C07332=1142.732,180.270,-61.153,-178.357,7.250,148.882
C07333=1142.727,180.518,-61.175,-178.354,7.252,148.881
C07334=1142.723,180.767,-61.199,-178.351,7.255,148.881
C07335=1142.718,181.017,-61.221,-178.348,7.256,148.881
C07336=1142.714,181.265,-61.244,-178.346,7.259,148.881
C07337=1142.709,181.514,-61.268,-178.343,7.261,148.880
C07338=1142.704,181.763,-61.291,-178.340,7.264,148.880
C07339=1142.700,182.011,-61.313,-178.337,7.266,148.880
C07340=1142.695,182.260,-61.337,-178.334,7.268,148.879
C07341=1142.690,182.509,-61.360,-178.332,7.270,148.879
C07342=1142.686,182.758,-61.383,-178.329,7.273,148.879
C07343=1142.682,183.007,-61.406,-178.326,7.275,148.879
C07344=1142.676,183.277,-61.431,-178.323,7.277,148.878
C07345=1142.671,183.547,-61.456,-178.320,7.280,148.878
C07346=1142.666,183.817,-61.481,-178.316,7.283,148.878
C07347=1142.661,184.085,-61.506,-178.314,7.285,148.878
C07348=1142.657,184.334,-61.530,-178.311,7.287,148.877
C07349=1142.652,184.583,-61.553,-178.308,7.290,148.877
C07350=1142.647,184.832,-61.576,-178.305,7.292,148.877
C07351=1142.643,185.081,-61.600,-178.302,7.294,148.876
C07352=1142.639,185.330,-61.623,-178.300,7.296,148.876
C07353=1142.634,185.579,-61.646,-178.297,7.299,148.876
C07354=1142.629,185.828,-61.669,-178.294,7.301,148.876
C07355=1142.625,186.077,-61.693,-178.291,7.304,148.875
C07356=1142.620,186.326,-61.716,-178.289,7.306,148.875
C07357=1142.615,186.575,-61.739,-178.286,7.308,148.875
C07358=1142.612,186.823,-61.763,-178.283,7.311,148.875
C07359=1142.607,187.072,-61.786,-178.280,7.313,148.874
C07360=1142.602,187.321,-61.809,-178.277,7.315,148.874
C07361=1142.597,187.570,-61.833,-178.275,7.318,148.874
C07362=1142.592,187.819,-61.856,-178.271,7.320,148.874
C07363=1142.587,188.068,-61.879,-178.269,7.322,148.874
C07364=1142.583,188.316,-61.903,-178.266,7.325,148.873
C07365=1142.578,188.565,-61.927,-178.264,7.327,148.873
C07366=1142.574,188.814,-61.950,-178.260,7.329,148.873
C07367=1142.569,189.063,-61.973,-178.258,7.331,148.873
C07368=1142.565,189.312,-61.998,-178.255,7.334,148.872
C07369=1142.560,189.561,-62.021,-178.252,7.337,148.872
C07370=1142.555,189.810,-62.044,-178.249,7.339,148.872
C07371=1142.551,190.058,-62.068,-178.247,7.342,148.872
C07372=1142.546,190.307,-62.092,-178.244,7.343,148.871
C07373=1142.541,190.556,-62.115,-178.241,7.346,148.871
C07374=1142.537,190.805,-62.139,-178.238,7.348,148.871
C07375=1142.532,191.054,-62.162,-178.236,7.351,148.871
C07376=1142.528,191.303,-62.186,-178.232,7.353,148.870
C07377=1142.523,191.551,-62.210,-178.230,7.355,148.870
C07378=1142.518,191.800,-62.233,-178.227,7.358,148.870
C07379=1142.514,192.050,-62.257,-178.224,7.360,148.870
C07380=1142.510,192.298,-62.281,-178.221,7.363,148.869
C07381=1142.505,192.547,-62.304,-178.218,7.366,148.869
C07382=1142.501,192.796,-62.328,-178.216,7.367,148.869
C07383=1142.496,193.045,-62.352,-178.213,7.370,148.869
C07384=1142.492,193.293,-62.376,-178.210,7.372,148.868
C07385=1142.487,193.542,-62.399,-178.207,7.375,148.868
C07386=1142.482,193.791,-62.424,-178.205,7.377,148.868
C07387=1142.477,194.040,-62.447,-178.202,7.379,148.868
C07388=1142.473,194.289,-62.471,-178.199,7.382,148.868
C07389=1142.468,194.538,-62.495,-178.196,7.384,148.867
C07390=1142.464,194.786,-62.519,-178.193,7.387,148.867
C07391=1142.460,195.036,-62.543,-178.190,7.390,148.867
C07392=1142.455,195.284,-62.567,-178.188,7.391,148.867
C07393=1142.450,195.533,-62.591,-178.185,7.394,148.866
C07394=1142.445,195.782,-62.615,-178.182,7.396,148.866
C07395=1142.441,196.030,-62.639,-178.179,7.399,148.866
C07396=1142.436,196.279,-62.662,-178.176,7.401,148.866
C07397=1142.432,196.528,-62.686,-178.174,7.403,148.866
C07398=1142.428,196.777,-62.711,-178.171,7.406,148.865
C07399=1142.423,197.026,-62.735,-178.168,7.408,148.865
C07400=1142.418,197.275,-62.759,-178.166,7.411,148.865
C07401=1142.414,197.523,-62.783,-178.162,7.414,148.865
C07402=1142.409,197.772,-62.806,-178.160,7.416,148.865
C07403=1142.404,198.021,-62.831,-178.157,7.418,148.864
C07404=1142.400,198.270,-62.855,-178.154,7.421,148.864
C07405=1142.396,198.519,-62.879,-178.151,7.423,148.864
C07406=1142.391,198.767,-62.903,-178.148,7.426,148.864
C07407=1142.386,199.016,-62.927,-178.146,7.427,148.863
C07408=1142.382,199.264,-62.951,-178.143,7.430,148.863
C07409=1142.378,199.514,-62.976,-178.140,7.433,148.863
C07410=1142.372,199.763,-63.000,-178.137,7.435,148.863
C07411=1142.368,200.011,-63.024,-178.135,7.438,148.863
C07412=1142.364,200.260,-63.048,-178.131,7.440,148.862
C07413=1142.359,200.509,-63.073,-178.129,7.443,148.862
C07414=1142.355,200.758,-63.097,-178.126,7.445,148.862
C07415=1142.350,201.006,-63.121,-178.123,7.448,148.862
C07416=1142.345,201.255,-63.145,-178.121,7.450,148.862
C07417=1142.341,201.504,-63.169,-178.118,7.453,148.861
C07418=1142.337,201.753,-63.194,-178.115,7.456,148.861
C07419=1142.332,202.002,-63.218,-178.112,7.457,148.861
C07420=1142.327,202.250,-63.242,-178.109,7.460,148.861
C07421=1142.323,202.499,-63.267,-178.106,7.463,148.861
C07422=1142.318,202.748,-63.291,-178.104,7.465,148.860
C07423=1142.314,202.996,-63.315,-178.101,7.468,148.860
C07424=1142.309,203.246,-63.341,-178.098,7.470,148.860
C07425=1142.305,203.494,-63.365,-178.095,7.472,148.860
C07426=1142.300,203.743,-63.389,-178.093,7.475,148.860
C07427=1142.295,203.991,-63.413,-178.089,7.478,148.859
C07428=1142.292,204.240,-63.438,-178.087,7.480,148.859
C07429=1142.287,204.489,-63.462,-178.084,7.483,148.859
C07430=1142.282,204.737,-63.487,-178.081,7.485,148.859
C07431=1142.278,204.987,-63.512,-178.079,7.488,148.859
C07432=1142.273,205.235,-63.536,-178.076,7.490,148.858
C07433=1142.268,205.484,-63.560,-178.073,7.493,148.858
C07434=1142.264,205.733,-63.585,-178.071,7.495,148.858
C07435=1142.259,205.981,-63.610,-178.067,7.498,148.858
C07436=1142.254,206.230,-63.635,-178.064,7.501,148.858
C07437=1142.251,206.479,-63.659,-178.062,7.503,148.857
C07438=1142.245,206.728,-63.684,-178.059,7.505,148.857
C07439=1142.242,206.977,-63.708,-178.056,7.508,148.857
C07440=1142.236,207.226,-63.733,-178.053,7.511,148.857
C07441=1142.232,207.473,-63.758,-178.051,7.513,148.857
C07442=1142.228,207.723,-63.783,-178.048,7.516,148.856
C07443=1142.223,207.972,-63.807,-178.045,7.518,148.856
C07444=1142.218,208.220,-63.832,-178.042,7.520,148.856
C07445=1142.214,208.469,-63.857,-178.040,7.523,148.856
C07446=1142.210,208.717,-63.881,-178.036,7.526,148.856
C07447=1142.205,208.967,-63.906,-178.034,7.529,148.855
C07448=1142.200,209.237,-63.933,-178.031,7.532,148.855
C07449=1142.195,209.508,-63.960,-178.027,7.534,148.855
C07450=1142.190,209.778,-63.987,-178.025,7.537,148.855
C07451=1142.185,210.049,-64.015,-178.021,7.540,148.855
C07452=1142.181,210.297,-64.039,-178.019,7.543,148.855
C07453=1142.176,210.546,-64.064,-178.016,7.545,148.854
C07454=1142.171,210.795,-64.089,-178.013,7.547,148.854
C07455=1142.168,211.044,-64.114,-178.010,7.550,148.854
C07456=1142.163,211.292,-64.139,-178.008,7.552,148.854
C07457=1142.158,211.542,-64.164,-178.005,7.555,148.854
C07458=1142.154,211.789,-64.189,-178.002,7.558,148.853
C07459=1142.150,212.039,-64.214,-177.999,7.561,148.853
C07460=1142.145,212.287,-64.239,-177.996,7.562,148.853
C07461=1142.140,212.536,-64.264,-177.994,7.565,148.853
C07462=1142.136,212.784,-64.289,-177.991,7.568,148.853
C07463=1142.132,213.034,-64.314,-177.988,7.571,148.853
C07464=1142.127,213.282,-64.339,-177.985,7.573,148.852
C07465=1142.122,213.531,-64.364,-177.983,7.576,148.852
C07466=1142.117,213.779,-64.390,-177.980,7.579,148.852
C07467=1142.114,214.028,-64.414,-177.977,7.581,148.852
C07468=1142.109,214.276,-64.440,-177.974,7.583,148.852
C07469=1142.104,214.526,-64.465,-177.971,7.586,148.852
C07470=1142.099,214.774,-64.490,-177.969,7.589,148.851
C07471=1142.095,215.023,-64.515,-177.965,7.592,148.851
C07472=1142.091,215.271,-64.540,-177.963,7.595,148.851
C07473=1142.087,215.520,-64.566,-177.960,7.597,148.851
C07474=1142.082,215.769,-64.591,-177.958,7.600,148.851
C07475=1142.077,216.018,-64.616,-177.954,7.602,148.851
C07476=1142.073,216.266,-64.642,-177.952,7.605,148.850
C07477=1142.068,216.515,-64.667,-177.949,7.607,148.850
C07478=1142.064,216.764,-64.692,-177.947,7.610,148.850
C07479=1142.059,217.012,-64.718,-177.943,7.613,148.850
C07480=1142.055,217.261,-64.742,-177.940,7.615,148.850
C07481=1142.051,217.510,-64.768,-177.938,7.618,148.850
C07482=1142.046,217.758,-64.793,-177.935,7.620,148.850
C07483=1142.042,218.007,-64.819,-177.932,7.623,148.849
C07484=1142.037,218.256,-64.844,-177.929,7.626,148.849
C07485=1142.032,218.504,-64.869,-177.927,7.629,148.849
C07486=1142.028,218.753,-64.895,-177.924,7.631,148.849
C07487=1142.023,219.001,-64.921,-177.921,7.634,148.849
C07488=1142.019,219.251,-64.946,-177.918,7.636,148.849
C07489=1142.015,219.499,-64.971,-177.915,7.639,148.848
C07490=1142.010,219.748,-64.997,-177.913,7.642,148.848
C07491=1142.005,219.996,-65.022,-177.910,7.644,148.848
C07492=1142.001,220.245,-65.048,-177.907,7.647,148.848
C07493=1141.996,220.493,-65.074,-177.904,7.650,148.848
C07494=1141.992,220.742,-65.099,-177.902,7.653,148.848
C07495=1141.988,220.991,-65.125,-177.899,7.656,148.848
C07496=1141.983,221.240,-65.150,-177.896,7.658,148.847
C07497=1141.979,221.488,-65.175,-177.893,7.660,148.847
C07498=1141.974,221.737,-65.201,-177.890,7.663,148.847
C07499=1141.970,221.985,-65.227,-177.888,7.666,148.847
C07500=1141.965,222.234,-65.252,-177.885,7.669,148.847
C07501=1141.961,222.483,-65.278,-177.882,7.672,148.847
C07502=1141.956,222.732,-65.304,-177.879,7.674,148.847
C07503=1141.951,222.980,-65.330,-177.877,7.677,148.846
C07504=1141.947,223.229,-65.356,-177.874,7.680,148.846
C07505=1141.943,223.478,-65.381,-177.871,7.682,148.846
C07506=1141.939,223.727,-65.407,-177.868,7.685,148.846
C07507=1141.934,223.975,-65.433,-177.865,7.688,148.846
C07508=1141.930,224.223,-65.459,-177.863,7.690,148.846
C07509=1141.926,224.472,-65.485,-177.860,7.693,148.846
C07510=1141.921,224.721,-65.511,-177.857,7.696,148.846
C07511=1141.916,224.969,-65.536,-177.854,7.699,148.845
C07512=1141.912,225.218,-65.562,-177.851,7.701,148.845
C07513=1141.907,225.466,-65.588,-177.848,7.704,148.845
C07514=1141.903,225.715,-65.614,-177.845,7.707,148.845
C07515=1141.898,225.964,-65.640,-177.843,7.709,148.845
C07516=1141.894,226.212,-65.666,-177.840,7.712,148.845
C07517=1141.890,226.461,-65.692,-177.838,7.715,148.845
C07518=1141.885,226.710,-65.718,-177.834,7.718,148.844
C07519=1141.880,226.959,-65.744,-177.832,7.721,148.844
C07520=1141.876,227.207,-65.769,-177.829,7.723,148.844
C07521=1141.872,227.455,-65.796,-177.826,7.726,148.844
C07522=1141.867,227.704,-65.822,-177.824,7.728,148.844
C07523=1141.862,227.953,-65.848,-177.821,7.731,148.844
C07524=1141.858,228.201,-65.874,-177.818,7.734,148.844
C07525=1141.854,228.450,-65.900,-177.815,7.737,148.844
C07526=1141.849,228.698,-65.926,-177.812,7.740,148.843
C07527=1141.845,228.946,-65.953,-177.809,7.743,148.843
C07528=1141.841,229.195,-65.978,-177.807,7.746,148.843
C07529=1141.836,229.444,-66.004,-177.804,7.748,148.843
C07530=1141.832,229.693,-66.031,-177.802,7.751,148.843
C07531=1141.827,229.941,-66.057,-177.799,7.754,148.843
C07532=1141.822,230.190,-66.083,-177.796,7.756,148.843
C07533=1141.818,230.438,-66.109,-177.793,7.759,148.843
C07534=1141.814,230.687,-66.135,-177.790,7.762,148.842
C07535=1141.809,230.935,-66.162,-177.787,7.765,148.842
C07536=1141.805,231.184,-66.188,-177.784,7.768,148.842
C07537=1141.801,231.432,-66.214,-177.781,7.771,148.842
C07538=1141.796,231.681,-66.241,-177.779,7.773,148.842
C07539=1141.792,231.930,-66.266,-177.776,7.776,148.842
C07540=1141.787,232.179,-66.294,-177.774,7.779,148.842
C07541=1141.783,232.427,-66.320,-177.771,7.782,148.842
C07542=1141.778,232.676,-66.346,-177.768,7.784,148.842
C07543=1141.774,232.924,-66.373,-177.765,7.787,148.841
C07544=1141.769,233.173,-66.399,-177.762,7.790,148.841
C07545=1141.765,233.421,-66.425,-177.759,7.793,148.841
C07546=1141.761,233.670,-66.451,-177.756,7.796,148.841
C07547=1141.756,233.918,-66.478,-177.754,7.799,148.841
C07548=1141.752,234.167,-66.504,-177.751,7.801,148.841
C07549=1141.747,234.415,-66.531,-177.749,7.804,148.841
C07550=1141.743,234.663,-66.557,-177.746,7.807,148.841
C07551=1141.738,234.913,-66.584,-177.743,7.810,148.841
C07552=1141.734,235.185,-66.613,-177.740,7.812,148.841
C07553=1141.729,235.456,-66.642,-177.736,7.816,148.840
C07554=1141.724,235.728,-66.671,-177.734,7.819,148.840
C07555=1141.719,236.000,-66.700,-177.731,7.822,148.840
C07556=1141.715,236.248,-66.727,-177.728,7.825,148.840
C07557=1141.710,236.497,-66.754,-177.725,7.827,148.840
C07558=1141.705,236.746,-66.780,-177.722,7.830,148.840
C07559=1141.701,236.994,-66.807,-177.720,7.833,148.840
C07560=1141.697,237.242,-66.834,-177.717,7.836,148.840
C07561=1141.693,237.491,-66.860,-177.714,7.839,148.840
C07562=1141.689,237.740,-66.887,-177.711,7.842,148.840
C07563=1141.684,237.989,-66.914,-177.708,7.845,148.840
C07564=1141.680,238.237,-66.940,-177.706,7.848,148.840
C07565=1141.675,238.486,-66.967,-177.702,7.850,148.839
C07566=1141.670,238.734,-66.994,-177.700,7.853,148.839
C07567=1141.667,238.982,-67.021,-177.697,7.856,148.839
C07568=1141.662,239.231,-67.048,-177.695,7.858,148.839
C07569=1141.657,239.480,-67.074,-177.692,7.861,148.839
C07570=1141.653,239.728,-67.101,-177.689,7.864,148.839
C07571=1141.648,239.977,-67.128,-177.686,7.867,148.839
C07572=1141.644,240.225,-67.155,-177.683,7.870,148.839
C07573=1141.639,240.474,-67.182,-177.681,7.873,148.839
C07574=1141.635,240.722,-67.208,-177.678,7.876,148.838
C07575=1141.631,240.971,-67.236,-177.675,7.879,148.838
C07576=1141.626,241.220,-67.263,-177.672,7.882,148.838
C07577=1141.622,241.468,-67.289,-177.669,7.885,148.838
C07578=1141.618,241.716,-67.316,-177.667,7.888,148.838
C07579=1141.613,241.965,-67.343,-177.664,7.890,148.838
C07580=1141.608,242.213,-67.371,-177.661,7.893,148.838
C07581=1141.604,242.462,-67.398,-177.658,7.896,148.838
C07582=1141.601,242.711,-67.424,-177.655,7.899,148.838
C07583=1141.596,242.959,-67.451,-177.653,7.902,148.838
C07584=1141.591,243.207,-67.479,-177.650,7.905,148.838
C07585=1141.587,243.455,-67.506,-177.647,7.908,148.838
C07586=1141.582,243.704,-67.533,-177.644,7.911,148.838
C07587=1141.578,243.952,-67.560,-177.641,7.914,148.837
C07588=1141.574,244.201,-67.587,-177.639,7.917,148.837
C07589=1141.570,244.450,-67.614,-177.636,7.920,148.837
C07590=1141.565,244.698,-67.641,-177.633,7.923,148.837
C07591=1141.561,244.946,-67.669,-177.630,7.925,148.837
C07592=1141.556,245.195,-67.696,-177.627,7.928,148.837
C07593=1141.552,245.444,-67.724,-177.625,7.931,148.837
C07594=1141.547,245.692,-67.751,-177.622,7.934,148.837
C07595=1141.543,245.940,-67.779,-177.619,7.937,148.837
C07596=1141.538,246.189,-67.806,-177.616,7.940,148.837
C07597=1141.534,246.437,-67.832,-177.613,7.943,148.837
C07598=1141.530,246.686,-67.859,-177.611,7.946,148.837
C07599=1141.526,246.934,-67.887,-177.608,7.949,148.837
C07600=1141.521,247.182,-67.914,-177.606,7.952,148.837
C07601=1141.517,247.431,-67.941,-177.603,7.955,148.837
C07602=1141.513,247.680,-67.970,-177.600,7.958,148.837
C07603=1141.508,247.928,-67.997,-177.597,7.961,148.836
C07604=1141.503,248.177,-68.024,-177.594,7.964,148.836
C07605=1141.499,248.424,-68.051,-177.592,7.967,148.836
C07606=1141.495,248.674,-68.079,-177.589,7.970,148.836
C07607=1141.491,248.921,-68.107,-177.586,7.973,148.836
C07608=1141.486,249.170,-68.134,-177.583,7.975,148.836
C07609=1141.482,249.419,-68.161,-177.580,7.978,148.836
C07610=1141.478,249.667,-68.189,-177.578,7.981,148.836
C07611=1141.473,249.916,-68.216,-177.575,7.984,148.836
C07612=1141.469,250.164,-68.245,-177.572,7.987,148.836
C07613=1141.464,250.413,-68.272,-177.569,7.990,148.836
C07614=1141.459,250.661,-68.300,-177.566,7.993,148.836
C07615=1141.455,250.910,-68.327,-177.564,7.996,148.836
C07616=1141.451,251.158,-68.355,-177.561,7.999,148.836
C07617=1141.446,251.406,-68.382,-177.558,8.002,148.836
C07618=1141.443,251.655,-68.410,-177.556,8.005,148.836
C07619=1141.438,251.903,-68.438,-177.553,8.008,148.836
C07620=1141.434,252.151,-68.465,-177.550,8.011,148.835
C07621=1141.430,252.400,-68.493,-177.547,8.014,148.835
C07622=1141.425,252.649,-68.521,-177.545,8.017,148.835
C07623=1141.420,252.897,-68.548,-177.542,8.020,148.835
C07624=1141.416,253.145,-68.576,-177.539,8.022,148.835
C07625=1141.412,253.394,-68.604,-177.536,8.025,148.835
C07626=1141.408,253.642,-68.632,-177.533,8.028,148.835
C07627=1141.403,253.890,-68.660,-177.531,8.032,148.835
C07628=1141.398,254.139,-68.687,-177.528,8.035,148.835
C07629=1141.395,254.388,-68.715,-177.525,8.037,148.835
C07630=1141.390,254.635,-68.743,-177.523,8.040,148.835
C07631=1141.386,254.884,-68.771,-177.520,8.043,148.835
C07632=1141.381,255.133,-68.799,-177.517,8.046,148.835
C07633=1141.377,255.381,-68.827,-177.514,8.050,148.835
C07634=1141.373,255.629,-68.855,-177.511,8.053,148.835
C07635=1141.369,255.877,-68.883,-177.509,8.056,148.835
C07636=1141.364,256.127,-68.911,-177.506,8.059,148.835
C07637=1141.359,256.374,-68.938,-177.503,8.062,148.835
C07638=1141.356,256.623,-68.966,-177.500,8.065,148.835
C07639=1141.351,256.871,-68.995,-177.497,8.068,148.835
C07640=1141.347,257.120,-69.023,-177.495,8.071,148.835
C07641=1141.343,257.368,-69.051,-177.492,8.074,148.834
C07642=1141.338,257.617,-69.080,-177.489,8.077,148.835
C07643=1141.334,257.864,-69.107,-177.487,8.080,148.835
C07644=1141.330,258.114,-69.135,-177.484,8.083,148.834
C07645=1141.325,258.362,-69.163,-177.481,8.086,148.834
C07646=1141.321,258.610,-69.191,-177.478,8.089,148.834
C07647=1141.316,258.858,-69.219,-177.475,8.092,148.834
C07648=1141.312,259.107,-69.248,-177.472,8.095,148.834
C07649=1141.308,259.355,-69.276,-177.470,8.099,148.834
C07650=1141.303,259.604,-69.304,-177.467,8.101,148.834
C07651=1141.299,259.852,-69.332,-177.464,8.104,148.834
C07652=1141.295,260.100,-69.360,-177.461,8.107,148.834
C07653=1141.290,260.349,-69.389,-177.459,8.110,148.834
C07654=1141.286,260.597,-69.417,-177.456,8.113,148.834
C07655=1141.281,260.845,-69.445,-177.453,8.116,148.834
C07656=1141.277,261.119,-69.477,-177.450,8.120,148.834
C07657=1141.272,261.392,-69.508,-177.447,8.123,148.834
C07658=1141.267,261.666,-69.539,-177.444,8.127,148.834
C07659=1141.262,261.939,-69.570,-177.441,8.130,148.834
C07660=1141.258,262.187,-69.599,-177.438,8.133,148.834
C07661=1141.254,262.436,-69.628,-177.436,8.136,148.834
C07662=1141.250,262.684,-69.655,-177.433,8.139,148.834
C07663=1141.245,262.933,-69.684,-177.430,8.143,148.834
C07664=1141.241,263.181,-69.712,-177.427,8.145,148.834
C07665=1141.237,263.429,-69.741,-177.424,8.148,148.834
C07666=1141.233,263.678,-69.770,-177.422,8.152,148.834
C07667=1141.228,263.926,-69.798,-177.419,8.155,148.834
C07668=1141.224,264.174,-69.826,-177.416,8.157,148.834
C07669=1141.219,264.423,-69.854,-177.414,8.160,148.834
C07670=1141.215,264.671,-69.884,-177.411,8.163,148.834
C07671=1141.211,264.920,-69.912,-177.408,8.167,148.834
C07672=1141.206,265.168,-69.940,-177.405,8.170,148.834
C07673=1141.202,265.416,-69.969,-177.402,8.173,148.834
C07674=1141.198,265.665,-69.998,-177.399,8.176,148.834
C07675=1141.193,265.913,-70.026,-177.397,8.179,148.834
C07676=1141.189,266.161,-70.055,-177.394,8.182,148.834
C07677=1141.185,266.410,-70.084,-177.392,8.185,148.834
C07678=1141.180,266.657,-70.113,-177.389,8.188,148.834
C07679=1141.176,266.906,-70.141,-177.386,8.191,148.834
C07680=1141.172,267.155,-70.170,-177.383,8.195,148.834
C07681=1141.167,267.402,-70.199,-177.380,8.198,148.834
C07682=1141.163,267.651,-70.227,-177.377,8.201,148.834
C07683=1141.159,267.899,-70.257,-177.375,8.204,148.834
C07684=1141.155,268.148,-70.285,-177.372,8.207,148.834
C07685=1141.150,268.395,-70.314,-177.370,8.210,148.834
C07686=1141.146,268.644,-70.343,-177.367,8.213,148.834
C07687=1141.142,268.892,-70.372,-177.364,8.217,148.834
C07688=1141.137,269.140,-70.400,-177.361,8.220,148.834
C07689=1141.133,269.388,-70.429,-177.358,8.223,148.834
C07690=1141.129,269.637,-70.458,-177.356,8.226,148.834
C07691=1141.125,269.886,-70.487,-177.353,8.229,148.834
C07692=1141.120,270.133,-70.517,-177.350,8.232,148.834
C07693=1141.115,270.382,-70.545,-177.348,8.235,148.834
C07694=1141.112,270.630,-70.574,-177.345,8.239,148.834
C07695=1141.108,270.879,-70.603,-177.342,8.242,148.834
C07696=1141.103,271.126,-70.632,-177.339,8.245,148.834
C07697=1141.099,271.375,-70.661,-177.337,8.248,148.834
C07698=1141.094,271.624,-70.690,-177.334,8.251,148.834
C07699=1141.090,271.872,-70.720,-177.331,8.254,148.834
C07700=1141.086,272.120,-70.748,-177.328,8.258,148.834
C07701=1141.081,272.368,-70.777,-177.325,8.261,148.834
C07702=1141.077,272.616,-70.806,-177.323,8.264,148.834
C07703=1141.073,272.865,-70.836,-177.320,8.267,148.834
C07704=1141.069,273.113,-70.865,-177.318,8.270,148.834
C07705=1141.064,273.362,-70.894,-177.315,8.273,148.834
C07706=1141.060,273.610,-70.923,-177.311,8.277,148.834
C07707=1141.055,273.858,-70.952,-177.309,8.280,148.834
C07708=1141.051,274.106,-70.982,-177.306,8.283,148.834
C07709=1141.048,274.354,-71.011,-177.303,8.286,148.834
C07710=1141.044,274.602,-71.040,-177.301,8.289,148.834
C07711=1141.039,274.851,-71.069,-177.298,8.292,148.834
C07712=1141.035,275.099,-71.098,-177.295,8.296,148.834
C07713=1141.031,275.347,-71.128,-177.293,8.299,148.834
C07714=1141.027,275.596,-71.157,-177.290,8.302,148.834
C07715=1141.022,275.843,-71.186,-177.288,8.305,148.834
C07716=1141.018,276.092,-71.216,-177.285,8.308,148.834
C07717=1141.013,276.340,-71.245,-177.281,8.312,148.834
C07718=1141.009,276.588,-71.275,-177.279,8.315,148.835
C07719=1141.005,276.836,-71.304,-177.276,8.318,148.835
C07720=1141.001,277.085,-71.334,-177.273,8.321,148.834
C07721=1140.997,277.333,-71.363,-177.271,8.324,148.835
C07722=1140.992,277.581,-71.393,-177.268,8.328,148.835
C07723=1140.988,277.829,-71.422,-177.265,8.331,148.835
C07724=1140.984,278.078,-71.452,-177.263,8.334,148.835
C07725=1140.979,278.326,-71.482,-177.260,8.337,148.835
C07726=1140.975,278.575,-71.511,-177.257,8.340,148.835
C07727=1140.971,278.823,-71.540,-177.254,8.344,148.835
C07728=1140.966,279.070,-71.570,-177.251,8.347,148.835
C07729=1140.962,279.319,-71.599,-177.249,8.350,148.835
C07730=1140.958,279.567,-71.628,-177.246,8.353,148.835
C07731=1140.954,279.815,-71.659,-177.244,8.357,148.835
C07732=1140.950,280.063,-71.688,-177.240,8.360,148.835
C07733=1140.945,280.311,-71.718,-177.238,8.363,148.835
C07734=1140.941,280.560,-71.748,-177.235,8.367,148.835
C07735=1140.936,280.808,-71.777,-177.233,8.369,148.835
C07736=1140.932,281.056,-71.806,-177.230,8.373,148.835
C07737=1140.928,281.304,-71.837,-177.227,8.376,148.835
C07738=1140.924,281.552,-71.866,-177.225,8.380,148.835
C07739=1140.919,281.801,-71.896,-177.222,8.383,148.835
C07740=1140.915,282.049,-71.926,-177.219,8.386,148.835
C07741=1140.911,282.297,-71.956,-177.216,8.390,148.835
C07742=1140.907,282.545,-71.985,-177.213,8.393,148.835
C07743=1140.902,282.793,-72.015,-177.211,8.396,148.836
C07744=1140.898,283.041,-72.045,-177.208,8.399,148.836
C07745=1140.895,283.290,-72.075,-177.205,8.403,148.836
C07746=1140.890,283.538,-72.105,-177.202,8.406,148.836
C07747=1140.886,283.786,-72.135,-177.200,8.409,148.836
C07748=1140.882,284.035,-72.165,-177.197,8.412,148.836
C07749=1140.877,284.283,-72.194,-177.195,8.415,148.836
C07750=1140.873,284.531,-72.225,-177.192,8.419,148.836
C07751=1140.869,284.779,-72.255,-177.189,8.422,148.836
C07752=1140.865,285.027,-72.285,-177.186,8.425,148.836
C07753=1140.860,285.275,-72.315,-177.184,8.428,148.836
C07754=1140.856,285.523,-72.345,-177.181,8.432,148.836
C07755=1140.852,285.771,-72.374,-177.178,8.435,148.836
C07756=1140.847,286.019,-72.405,-177.176,8.438,148.836
C07757=1140.844,286.268,-72.435,-177.173,8.441,148.836
C07758=1140.840,286.516,-72.465,-177.170,8.445,148.837
C07759=1140.835,286.764,-72.495,-177.167,8.448,148.836
C07760=1140.830,287.039,-72.529,-177.164,8.452,148.837
C07761=1140.825,287.316,-72.562,-177.161,8.455,148.837
C07762=1140.820,287.590,-72.595,-177.159,8.459,148.837
C07763=1140.816,287.866,-72.629,-177.155,8.463,148.837
C07764=1140.811,288.114,-72.659,-177.153,8.466,148.837
C07765=1140.808,288.362,-72.689,-177.150,8.469,148.837
C07766=1140.804,288.611,-72.720,-177.147,8.473,148.837
C07767=1140.799,288.859,-72.750,-177.144,8.476,148.837
C07768=1140.795,289.107,-72.781,-177.142,8.480,148.837
C07769=1140.791,289.355,-72.811,-177.139,8.483,148.837
C07770=1140.786,289.603,-72.841,-177.136,8.487,148.837
C07771=1140.783,289.851,-72.871,-177.133,8.489,148.837
C07772=1140.778,290.099,-72.902,-177.131,8.493,148.838
C07773=1140.774,290.348,-72.932,-177.128,8.496,148.838
C07774=1140.769,290.596,-72.962,-177.125,8.500,148.838
C07775=1140.765,290.843,-72.993,-177.123,8.503,148.838
C07776=1140.761,291.092,-73.024,-177.120,8.507,148.838
C07777=1140.758,291.340,-73.054,-177.117,8.510,148.838
C07778=1140.753,291.588,-73.084,-177.115,8.513,148.838
C07779=1140.749,291.836,-73.114,-177.112,8.516,148.838
C07780=1140.745,292.084,-73.145,-177.109,8.520,148.838
C07781=1140.741,292.332,-73.175,-177.107,8.523,148.838
C07782=1140.736,292.580,-73.206,-177.104,8.526,148.839
C07783=1140.732,292.828,-73.237,-177.101,8.530,148.839
C07784=1140.728,293.076,-73.267,-177.099,8.533,148.839
C07785=1140.723,293.325,-73.298,-177.096,8.536,148.839
C07786=1140.719,293.573,-73.328,-177.093,8.540,148.839
C07787=1140.715,293.821,-73.358,-177.090,8.544,148.839
C07788=1140.711,294.069,-73.390,-177.088,8.547,148.839
C07789=1140.707,294.317,-73.420,-177.085,8.550,148.839
C07790=1140.702,294.565,-73.451,-177.082,8.554,148.839
C07791=1140.698,294.814,-73.482,-177.080,8.557,148.839
C07792=1140.695,295.061,-73.512,-177.077,8.560,148.840
C07793=1140.690,295.309,-73.543,-177.074,8.564,148.840
C07794=1140.686,295.558,-73.574,-177.072,8.567,148.840
C07795=1140.681,295.806,-73.604,-177.069,8.570,148.840
C07796=1140.677,296.053,-73.635,-177.066,8.574,148.840
C07797=1140.674,296.301,-73.666,-177.064,8.577,148.840
C07798=1140.669,296.549,-73.697,-177.061,8.580,148.840
C07799=1140.665,296.797,-73.727,-177.058,8.584,148.840
C07800=1140.661,297.046,-73.759,-177.056,8.588,148.840
C07801=1140.657,297.294,-73.789,-177.053,8.591,148.840
C07802=1140.653,297.542,-73.820,-177.050,8.595,148.841
C07803=1140.648,297.790,-73.851,-177.047,8.598,148.841
C07804=1140.644,298.037,-73.882,-177.045,8.601,148.841
C07805=1140.640,298.286,-73.913,-177.042,8.605,148.841
C07806=1140.636,298.534,-73.944,-177.039,8.608,148.841
C07807=1140.631,298.782,-73.975,-177.037,8.611,148.841
C07808=1140.627,299.031,-74.006,-177.034,8.615,148.841
C07809=1140.623,299.278,-74.037,-177.031,8.619,148.841
C07810=1140.620,299.526,-74.068,-177.029,8.621,148.841
C07811=1140.615,299.774,-74.099,-177.026,8.626,148.842
C07812=1140.611,300.021,-74.130,-177.023,8.629,148.842
C07813=1140.607,300.270,-74.161,-177.021,8.632,148.842
C07814=1140.602,300.518,-74.192,-177.018,8.636,148.842
C07815=1140.598,300.766,-74.224,-177.015,8.639,148.842
C07816=1140.594,301.014,-74.255,-177.013,8.642,148.842
C07817=1140.590,301.263,-74.286,-177.010,8.646,148.842
C07818=1140.585,301.510,-74.317,-177.007,8.649,148.842
C07819=1140.581,301.759,-74.348,-177.004,8.653,148.843
C07820=1140.577,302.007,-74.379,-177.002,8.656,148.843
C07821=1140.574,302.254,-74.410,-176.999,8.660,148.843
C07822=1140.569,302.502,-74.441,-176.996,8.664,148.843
C07823=1140.565,302.750,-74.473,-176.994,8.667,148.843
C07824=1140.561,302.998,-74.504,-176.991,8.670,148.843
C07825=1140.557,303.246,-74.535,-176.988,8.674,148.843
C07826=1140.553,303.494,-74.566,-176.986,8.677,148.844
C07827=1140.548,303.742,-74.598,-176.983,8.681,148.844
C07828=1140.544,303.991,-74.630,-176.980,8.684,148.844
C07829=1140.539,304.238,-74.661,-176.978,8.687,148.844
C07830=1140.535,304.487,-74.692,-176.975,8.692,148.844
C07831=1140.531,304.734,-74.724,-176.973,8.695,148.844
C07832=1140.527,304.983,-74.755,-176.970,8.698,148.844
C07833=1140.523,305.231,-74.787,-176.967,8.702,148.845
C07834=1140.519,305.478,-74.818,-176.965,8.705,148.845
C07835=1140.515,305.727,-74.849,-176.962,8.709,148.845
C07836=1140.511,305.974,-74.881,-176.959,8.712,148.845
C07837=1140.507,306.222,-74.913,-176.956,8.715,148.845
C07838=1140.502,306.470,-74.943,-176.954,8.719,148.845
C07839=1140.499,306.718,-74.975,-176.951,8.723,148.845
C07840=1140.493,306.966,-75.007,-176.948,8.727,148.846
C07841=1140.489,307.214,-75.038,-176.946,8.730,148.846
C07842=1140.486,307.462,-75.070,-176.943,8.733,148.846
C07843=1140.481,307.710,-75.102,-176.940,8.737,148.846
C07844=1140.478,307.958,-75.134,-176.938,8.740,148.846
C07845=1140.473,308.206,-75.164,-176.935,8.744,148.846
C07846=1140.469,308.454,-75.197,-176.932,8.747,148.846
C07847=1140.465,308.702,-75.229,-176.930,8.751,148.847
C07848=1140.461,308.950,-75.260,-176.927,8.755,148.847
C07849=1140.457,309.198,-75.292,-176.925,8.758,148.847
C07850=1140.452,309.446,-75.323,-176.922,8.762,148.847
C07851=1140.448,309.694,-75.355,-176.919,8.765,148.847
C07852=1140.444,309.942,-75.387,-176.917,8.768,148.847
C07853=1140.440,310.189,-75.418,-176.914,8.772,148.848
C07854=1140.436,310.437,-75.450,-176.911,8.775,148.848
C07855=1140.432,310.686,-75.483,-176.908,8.780,148.848
C07856=1140.427,310.933,-75.514,-176.906,8.783,148.848
C07857=1140.424,311.181,-75.546,-176.903,8.787,148.848
C07858=1140.419,311.429,-75.579,-176.901,8.790,148.849
C07859=1140.415,311.677,-75.610,-176.898,8.793,148.849
C07860=1140.411,311.925,-75.642,-176.895,8.797,148.849
C07861=1140.408,312.173,-75.674,-176.893,8.800,148.849
C07862=1140.403,312.421,-75.706,-176.890,8.804,148.849
C07863=1140.399,312.668,-75.738,-176.887,8.808,148.849
C07864=1140.394,312.946,-75.774,-176.885,8.812,148.850
C07865=1140.390,313.225,-75.810,-176.882,8.816,148.850
C07866=1140.385,313.503,-75.845,-176.879,8.820,148.850
C07867=1140.380,313.781,-75.881,-176.876,8.824,148.850
C07868=1140.377,314.029,-75.913,-176.873,8.828,148.850
C07869=1140.372,314.276,-75.946,-176.870,8.831,148.850
C07870=1140.368,314.524,-75.977,-176.868,8.834,148.851
C07871=1140.364,314.772,-76.010,-176.865,8.838,148.851
C07872=1140.360,315.020,-76.042,-176.862,8.842,148.851
C07873=1140.356,315.268,-76.074,-176.860,8.846,148.851
C07874=1140.352,315.515,-76.106,-176.857,8.849,148.851
C07875=1140.348,315.763,-76.138,-176.854,8.853,148.852
C07876=1140.343,316.011,-76.171,-176.852,8.856,148.852
C07877=1140.340,316.260,-76.202,-176.849,8.860,148.852
C07878=1140.335,316.507,-76.234,-176.847,8.864,148.852
C07879=1140.331,316.755,-76.267,-176.844,8.868,148.852
C07880=1140.327,317.003,-76.299,-176.841,8.871,148.853
C07881=1140.323,317.251,-76.331,-176.839,8.874,148.853
C07882=1140.319,317.499,-76.364,-176.836,8.878,148.853
C07883=1140.315,317.747,-76.396,-176.834,8.882,148.853
C07884=1140.310,317.994,-76.428,-176.831,8.886,148.853
C07885=1140.307,318.242,-76.461,-176.829,8.889,148.854
C07886=1140.302,318.490,-76.493,-176.826,8.893,148.854
C07887=1140.299,318.738,-76.526,-176.823,8.896,148.854
C07888=1140.295,318.986,-76.558,-176.820,8.900,148.854
C07889=1140.290,319.234,-76.591,-176.818,8.904,148.854
C07890=1140.286,319.481,-76.623,-176.815,8.908,148.855
C07891=1140.282,319.729,-76.655,-176.813,8.911,148.855
C07892=1140.278,319.977,-76.688,-176.810,8.915,148.855
C07893=1140.274,320.225,-76.720,-176.807,8.918,148.855
C07894=1140.270,320.473,-76.754,-176.805,8.922,148.856
C07895=1140.266,320.721,-76.785,-176.802,8.926,148.856
C07896=1140.262,320.969,-76.819,-176.799,8.930,148.856
C07897=1140.258,321.217,-76.850,-176.797,8.933,148.856
C07898=1140.254,321.464,-76.884,-176.794,8.937,148.856
C07899=1140.250,321.713,-76.916,-176.792,8.940,148.857
C07900=1140.246,321.960,-76.949,-176.789,8.944,148.857
C07901=1140.241,322.207,-76.981,-176.786,8.948,148.857
C07902=1140.237,322.456,-77.014,-176.783,8.952,148.857
C07903=1140.234,322.703,-77.046,-176.781,8.955,148.857
C07904=1140.229,322.951,-77.080,-176.778,8.959,148.858
C07905=1140.225,323.199,-77.112,-176.776,8.962,148.858
C07906=1140.221,323.447,-77.145,-176.773,8.966,148.858
C07907=1140.217,323.694,-77.178,-176.771,8.970,148.858
C07908=1140.213,323.943,-77.210,-176.768,8.974,148.859
C07909=1140.209,324.190,-77.243,-176.766,8.977,148.859
C07910=1140.205,324.438,-77.277,-176.763,8.981,148.859
C07911=1140.201,324.686,-77.308,-176.760,8.984,148.859
C07912=1140.197,324.934,-77.342,-176.758,8.989,148.860
C07913=1140.193,325.181,-77.375,-176.755,8.992,148.860
C07914=1140.189,325.429,-77.408,-176.752,8.996,148.860
C07915=1140.185,325.677,-77.441,-176.750,8.999,148.860
C07916=1140.181,325.925,-77.473,-176.747,9.003,148.860
C07917=1140.177,326.173,-77.506,-176.745,9.006,148.861
C07918=1140.173,326.420,-77.539,-176.742,9.011,148.861
C07919=1140.168,326.668,-77.572,-176.739,9.015,148.861
C07920=1140.164,326.916,-77.605,-176.737,9.018,148.861
C07921=1140.160,327.164,-77.639,-176.734,9.022,148.862
C07922=1140.156,327.411,-77.672,-176.732,9.026,148.862
C07923=1140.153,327.659,-77.704,-176.729,9.030,148.862
C07924=1140.148,327.907,-77.737,-176.726,9.033,148.862
C07925=1140.144,328.154,-77.771,-176.724,9.037,148.863
C07926=1140.140,328.403,-77.803,-176.722,9.041,148.863
C07927=1140.136,328.651,-77.837,-176.719,9.045,148.863
C07928=1140.132,328.899,-77.870,-176.716,9.048,148.863
C07929=1140.128,329.146,-77.903,-176.713,9.052,148.864
C07930=1140.124,329.394,-77.936,-176.710,9.056,148.864
C07931=1140.120,329.641,-77.970,-176.708,9.060,148.864
C07932=1140.116,329.889,-78.003,-176.706,9.064,148.864
C07933=1140.112,330.137,-78.036,-176.703,9.067,148.865
C07934=1140.108,330.385,-78.069,-176.700,9.071,148.865
C07935=1140.104,330.632,-78.103,-176.698,9.074,148.865
C07936=1140.099,330.880,-78.136,-176.695,9.079,148.865
C07937=1140.095,331.128,-78.169,-176.693,9.083,148.866
C07938=1140.092,331.376,-78.202,-176.690,9.086,148.866
C07939=1140.088,331.624,-78.236,-176.687,9.090,148.866
C07940=1140.084,331.871,-78.269,-176.685,9.093,148.866
C07941=1140.080,332.119,-78.303,-176.682,9.098,148.867
C07942=1140.075,332.366,-78.336,-176.680,9.101,148.867
C07943=1140.071,332.614,-78.369,-176.677,9.105,148.867
C07944=1140.068,332.863,-78.402,-176.674,9.109,148.867
C07945=1140.064,333.110,-78.436,-176.672,9.113,148.868
C07946=1140.060,333.357,-78.469,-176.669,9.117,148.868
C07947=1140.055,333.605,-78.503,-176.667,9.120,148.868
C07948=1140.051,333.853,-78.537,-176.664,9.124,148.868
C07949=1140.047,334.100,-78.570,-176.662,9.128,148.869
C07950=1140.043,334.349,-78.604,-176.659,9.132,148.869
C07951=1140.040,334.596,-78.638,-176.656,9.136,148.869
C07952=1140.035,334.844,-78.671,-176.654,9.139,148.870
C07953=1140.031,335.091,-78.704,-176.652,9.143,148.870
C07954=1140.027,335.339,-78.738,-176.649,9.147,148.870
C07955=1140.023,335.587,-78.772,-176.646,9.151,148.870
C07956=1140.019,335.835,-78.805,-176.644,9.155,148.871
C07957=1140.015,336.082,-78.839,-176.641,9.158,148.871
C07958=1140.011,336.330,-78.872,-176.638,9.162,148.871
C07959=1140.007,336.578,-78.907,-176.636,9.166,148.872
C07960=1140.003,336.826,-78.940,-176.634,9.170,148.872
C07961=1139.999,337.073,-78.974,-176.631,9.174,148.872
C07962=1139.995,337.320,-79.007,-176.628,9.177,148.872
C07963=1139.991,337.569,-79.042,-176.626,9.182,148.873
C07964=1139.987,337.816,-79.075,-176.624,9.185,148.873
C07965=1139.983,338.063,-79.109,-176.621,9.189,148.873
C07966=1139.980,338.312,-79.142,-176.618,9.194,148.874
C07967=1139.975,338.559,-79.177,-176.616,9.197,148.874
C07968=1139.971,338.840,-79.215,-176.612,9.202,148.874
C07969=1139.966,339.120,-79.253,-176.610,9.206,148.875
C07970=1139.962,339.401,-79.292,-176.607,9.210,148.875
C07971=1139.957,339.681,-79.330,-176.604,9.215,148.875
C07972=1139.954,339.929,-79.365,-176.601,9.219,148.876
C07973=1139.949,340.177,-79.398,-176.598,9.223,148.876
C07974=1139.945,340.424,-79.432,-176.597,9.226,148.876
C07975=1139.941,340.672,-79.467,-176.594,9.230,148.876
C07976=1139.937,340.920,-79.500,-176.592,9.234,148.877
C07977=1139.933,341.167,-79.534,-176.589,9.238,148.877
C07978=1139.929,341.415,-79.569,-176.586,9.242,148.877
C07979=1139.925,341.662,-79.603,-176.584,9.246,148.878
C07980=1139.920,341.911,-79.636,-176.581,9.250,148.878
C07981=1139.917,342.158,-79.671,-176.578,9.254,148.878
C07982=1139.912,342.406,-79.705,-176.576,9.257,148.879
C07983=1139.909,342.653,-79.739,-176.573,9.261,148.879
C07984=1139.905,342.901,-79.773,-176.571,9.266,148.879
C07985=1139.900,343.149,-79.807,-176.568,9.269,148.880
C07986=1139.897,343.397,-79.841,-176.566,9.273,148.880
C07987=1139.893,343.644,-79.876,-176.563,9.278,148.880
C07988=1139.889,343.891,-79.910,-176.561,9.281,148.880
C07989=1139.885,344.139,-79.944,-176.558,9.285,148.881
C07990=1139.881,344.386,-79.978,-176.555,9.289,148.881
C07991=1139.877,344.634,-80.013,-176.553,9.293,148.882
C07992=1139.872,344.882,-80.048,-176.550,9.297,148.882
C07993=1139.869,345.130,-80.082,-176.548,9.301,148.882
C07994=1139.865,345.377,-80.116,-176.545,9.305,148.882
C07995=1139.861,345.624,-80.150,-176.543,9.309,148.883
C07996=1139.857,345.872,-80.185,-176.540,9.313,148.883
C07997=1139.853,346.119,-80.219,-176.538,9.317,148.884
C07998=1139.849,346.368,-80.254,-176.535,9.321,148.884
C07999=1139.845,346.615,-80.288,-176.532,9.325,148.884
C08000=1139.841,346.863,-80.322,-176.530,9.328,148.884
C08001=1139.837,347.110,-80.357,-176.527,9.332,148.885
C08002=1139.833,347.358,-80.391,-176.525,9.337,148.885
C08003=1139.829,347.605,-80.426,-176.523,9.340,148.885
C08004=1139.825,347.854,-80.460,-176.520,9.344,148.886
C08005=1139.821,348.100,-80.495,-176.517,9.349,148.886
C08006=1139.817,348.348,-80.530,-176.515,9.352,148.886
C08007=1139.813,348.596,-80.564,-176.512,9.356,148.887
C08008=1139.810,348.843,-80.599,-176.510,9.361,148.887
C08009=1139.805,349.091,-80.633,-176.508,9.364,148.888
C08010=1139.801,349.338,-80.669,-176.505,9.368,148.888
C08011=1139.798,349.585,-80.702,-176.502,9.373,148.888
C08012=1139.794,349.834,-80.737,-176.499,9.377,148.888
C08013=1139.789,350.081,-80.772,-176.498,9.380,148.889
C08014=1139.785,350.328,-80.807,-176.495,9.384,148.889
C08015=1139.782,350.576,-80.842,-176.492,9.389,148.890
C08016=1139.778,350.824,-80.876,-176.490,9.392,148.890
C08017=1139.774,351.071,-80.912,-176.487,9.396,148.890
C08018=1139.769,351.319,-80.946,-176.484,9.400,148.890
C08019=1139.766,351.566,-80.980,-176.482,9.405,148.891
C08020=1139.762,351.813,-81.015,-176.480,9.408,148.891
C08021=1139.758,352.061,-81.050,-176.477,9.412,148.892
C08022=1139.754,352.309,-81.086,-176.474,9.417,148.892
C08023=1139.750,352.556,-81.120,-176.472,9.420,148.892
C08024=1139.746,352.804,-81.155,-176.470,9.424,148.893
C08025=1139.743,353.052,-81.190,-176.467,9.429,148.893
C08026=1139.738,353.299,-81.225,-176.464,9.433,148.893
C08027=1139.735,353.546,-81.260,-176.462,9.436,148.894
C08028=1139.730,353.794,-81.295,-176.459,9.441,148.894
C08029=1139.726,354.041,-81.330,-176.457,9.445,148.895
C08030=1139.722,354.289,-81.365,-176.454,9.449,148.895
C08031=1139.718,354.536,-81.400,-176.452,9.453,148.895
C08032=1139.715,354.783,-81.435,-176.449,9.457,148.896
C08033=1139.711,355.032,-81.470,-176.447,9.461,148.896
C08034=1139.707,355.278,-81.505,-176.445,9.465,148.896
C08035=1139.703,355.527,-81.540,-176.442,9.469,148.897
C08036=1139.699,355.774,-81.575,-176.439,9.473,148.897
C08037=1139.695,356.021,-81.611,-176.437,9.477,148.897
C08038=1139.691,356.269,-81.645,-176.435,9.481,148.898
C08039=1139.687,356.516,-81.681,-176.432,9.485,148.898
C08040=1139.684,356.764,-81.717,-176.429,9.489,148.899
C08041=1139.679,357.011,-81.751,-176.426,9.494,148.899
C08042=1139.675,357.259,-81.787,-176.424,9.497,148.899
C08043=1139.672,357.506,-81.822,-176.422,9.501,148.900
C08044=1139.668,357.754,-81.857,-176.419,9.506,148.900
C08045=1139.664,358.001,-81.892,-176.416,9.510,148.900
C08046=1139.660,358.249,-81.928,-176.414,9.514,148.901
C08047=1139.656,358.496,-81.963,-176.412,9.518,148.901
C08048=1139.653,358.744,-81.999,-176.409,9.522,148.902
C08049=1139.648,358.991,-82.033,-176.407,9.526,148.902
C08050=1139.644,359.239,-82.069,-176.404,9.530,148.902
C08051=1139.641,359.486,-82.104,-176.401,9.535,148.903
C08052=1139.637,359.734,-82.140,-176.399,9.538,148.903
C08053=1139.633,359.980,-82.175,-176.396,9.542,148.903
C08054=1139.629,360.228,-82.211,-176.394,9.547,148.904
C08055=1139.625,360.476,-82.246,-176.391,9.551,148.904
C08056=1139.621,360.723,-82.282,-176.389,9.556,148.905
C08057=1139.617,360.971,-82.318,-176.386,9.560,148.905
C08058=1139.613,361.218,-82.353,-176.384,9.563,148.905
C08059=1139.609,361.465,-82.389,-176.381,9.568,148.906
C08060=1139.606,361.713,-82.424,-176.378,9.572,148.906
C08061=1139.602,361.960,-82.460,-176.376,9.576,148.907
C08062=1139.598,362.208,-82.495,-176.373,9.580,148.907
C08063=1139.594,362.455,-82.531,-176.370,9.585,148.907
C08064=1139.590,362.702,-82.567,-176.368,9.589,148.908
C08065=1139.586,362.950,-82.602,-176.365,9.593,148.908
C08066=1139.582,363.197,-82.638,-176.363,9.597,148.909
C08067=1139.579,363.445,-82.673,-176.360,9.602,148.909
C08068=1139.575,363.692,-82.709,-176.358,9.605,148.909
C08069=1139.571,363.940,-82.745,-176.355,9.609,148.910
C08070=1139.567,364.188,-82.780,-176.353,9.614,148.910
C08071=1139.564,364.434,-82.817,-176.350,9.618,148.911
C08072=1139.558,364.719,-82.857,-176.347,9.623,148.911
C08073=1139.554,365.003,-82.899,-176.343,9.628,148.911
C08074=1139.550,365.286,-82.939,-176.341,9.633,148.912
C08075=1139.545,365.570,-82.981,-176.338,9.638,148.912
C08076=1139.542,365.817,-83.017,-176.335,9.642,148.913
C08077=1139.538,366.064,-83.052,-176.332,9.646,148.913
C08078=1139.533,366.312,-83.089,-176.330,9.651,148.914
C08079=1139.530,366.560,-83.124,-176.327,9.655,148.914
C08080=1139.526,366.806,-83.160,-176.324,9.659,148.914
C08081=1139.522,367.054,-83.197,-176.322,9.663,148.915
C08082=1139.518,367.302,-83.232,-176.319,9.668,148.915
C08083=1139.515,367.549,-83.268,-176.316,9.672,148.915
C08084=1139.511,367.796,-83.305,-176.314,9.676,148.916
C08085=1139.507,368.043,-83.341,-176.311,9.681,148.916
C08086=1139.503,368.291,-83.377,-176.309,9.685,148.917
C08087=1139.499,368.539,-83.412,-176.306,9.689,148.917
C08088=1139.496,368.786,-83.449,-176.303,9.694,148.918
C08089=1139.491,369.033,-83.485,-176.301,9.698,148.918
C08090=1139.488,369.280,-83.521,-176.298,9.702,148.918
C08091=1139.484,369.528,-83.557,-176.295,9.706,148.919
C08092=1139.480,369.775,-83.594,-176.293,9.711,148.919
C08093=1139.476,370.023,-83.630,-176.290,9.715,148.920
C08094=1139.473,370.270,-83.666,-176.288,9.719,148.920
C08095=1139.468,370.517,-83.702,-176.285,9.724,148.920
C08096=1139.465,370.764,-83.738,-176.282,9.728,148.921
C08097=1139.461,371.011,-83.775,-176.280,9.732,148.921
C08098=1139.457,371.259,-83.811,-176.277,9.736,148.922
C08099=1139.453,371.506,-83.848,-176.275,9.741,148.922
C08100=1139.450,371.753,-83.884,-176.272,9.745,148.923
C08101=1139.445,372.001,-83.920,-176.270,9.749,148.923
C08102=1139.442,372.248,-83.956,-176.268,9.753,148.923
C08103=1139.438,372.495,-83.993,-176.265,9.757,148.924
C08104=1139.434,372.743,-84.030,-176.262,9.762,148.924
C08105=1139.431,372.990,-84.066,-176.260,9.766,148.925
C08106=1139.427,373.238,-84.103,-176.257,9.770,148.925
C08107=1139.423,373.485,-84.138,-176.255,9.775,148.926
C08108=1139.419,373.732,-84.175,-176.253,9.778,148.926
C08109=1139.415,373.979,-84.212,-176.250,9.782,148.926
C08110=1139.411,374.226,-84.248,-176.247,9.787,148.927
C08111=1139.407,374.473,-84.285,-176.245,9.791,148.927
C08112=1139.403,374.721,-84.321,-176.243,9.795,148.928
C08113=1139.400,374.969,-84.358,-176.240,9.799,148.928
C08114=1139.396,375.216,-84.395,-176.238,9.803,148.929
C08115=1139.392,375.463,-84.432,-176.235,9.808,148.929
C08116=1139.389,375.710,-84.468,-176.233,9.811,148.929
C08117=1139.384,375.957,-84.505,-176.231,9.816,148.930
C08118=1139.380,376.205,-84.542,-176.229,9.819,148.930
C08119=1139.377,376.451,-84.578,-176.226,9.824,148.931
C08120=1139.373,376.699,-84.615,-176.224,9.827,148.931
C08121=1139.369,376.947,-84.651,-176.222,9.832,148.932
C08122=1139.365,377.194,-84.688,-176.220,9.835,148.932
C08123=1139.362,377.441,-84.724,-176.217,9.840,148.933
C08124=1139.358,377.688,-84.761,-176.215,9.843,148.933
C08125=1139.354,377.936,-84.798,-176.213,9.847,148.933
C08126=1139.350,378.183,-84.835,-176.211,9.851,148.934
C08127=1139.347,378.430,-84.872,-176.209,9.855,148.934
C08128=1139.343,378.677,-84.909,-176.207,9.858,148.935
C08129=1139.339,378.924,-84.946,-176.205,9.863,148.935
C08130=1139.335,379.172,-84.983,-176.203,9.867,148.936
C08131=1139.331,379.419,-85.020,-176.201,9.870,148.936
C08132=1139.327,379.666,-85.057,-176.200,9.874,148.937
C08133=1139.324,379.913,-85.093,-176.198,9.878,148.937
C08134=1139.320,380.161,-85.130,-176.196,9.881,148.938
C08135=1139.316,380.408,-85.167,-176.194,9.885,148.938
C08136=1139.312,380.656,-85.204,-176.193,9.889,148.939
C08137=1139.308,380.902,-85.242,-176.191,9.892,148.939
C08138=1139.305,381.150,-85.279,-176.189,9.896,148.940
C08139=1139.301,381.397,-85.316,-176.188,9.899,148.940
C08140=1139.297,381.644,-85.352,-176.186,9.903,148.941
C08141=1139.293,381.891,-85.389,-176.185,9.907,148.941
C08142=1139.290,382.138,-85.427,-176.184,9.910,148.942
C08143=1139.286,382.386,-85.464,-176.182,9.913,148.942
C08144=1139.282,382.633,-85.501,-176.181,9.916,148.943
C08145=1139.278,382.880,-85.537,-176.180,9.919,148.943
C08146=1139.274,383.128,-85.575,-176.179,9.923,148.944
C08147=1139.270,383.375,-85.612,-176.178,9.926,148.945
C08148=1139.266,383.622,-85.649,-176.177,9.929,148.945
C08149=1139.263,383.870,-85.686,-176.176,9.932,148.946
C08150=1139.260,384.116,-85.723,-176.175,9.936,148.946
C08151=1139.256,384.363,-85.760,-176.174,9.939,148.947
C08152=1139.252,384.611,-85.797,-176.173,9.942,148.948
C08153=1139.248,384.858,-85.835,-176.173,9.945,148.948
C08154=1139.244,385.105,-85.872,-176.172,9.948,148.949
C08155=1139.240,385.352,-85.909,-176.172,9.951,148.949
C08156=1139.237,385.599,-85.947,-176.171,9.954,148.950
C08157=1139.233,385.846,-85.984,-176.171,9.956,148.951
C08158=1139.229,386.094,-86.020,-176.170,9.959,148.951
C08159=1139.226,386.341,-86.058,-176.170,9.962,148.952
C08160=1139.222,386.588,-86.095,-176.169,9.965,148.953
C08161=1139.217,386.835,-86.132,-176.169,9.968,148.953
C08162=1139.214,387.082,-86.170,-176.169,9.970,148.954
C08163=1139.210,387.330,-86.207,-176.169,9.973,148.955
C08164=1139.206,387.577,-86.244,-176.169,9.976,148.955
C08165=1139.203,387.824,-86.282,-176.169,9.979,148.956
C08166=1139.199,388.071,-86.318,-176.169,9.981,148.957
C08167=1139.195,388.318,-86.356,-176.169,9.984,148.957
C08168=1139.192,388.566,-86.393,-176.169,9.986,148.958
C08169=1139.188,388.812,-86.431,-176.169,9.989,148.959
C08170=1139.184,389.060,-86.468,-176.170,9.991,148.959
C08171=1139.180,389.307,-86.505,-176.170,9.993,148.960
C08172=1139.176,389.554,-86.543,-176.170,9.996,148.961
C08173=1139.173,389.802,-86.580,-176.171,9.999,148.962
C08174=1139.169,390.048,-86.617,-176.171,10.000,148.962
C08175=1139.165,390.296,-86.654,-176.171,10.003,148.963
C08176=1139.160,390.583,-86.697,-176.172,10.006,148.964
C08177=1139.156,390.871,-86.742,-176.172,10.009,148.965
C08178=1139.152,391.158,-86.784,-176.173,10.012,148.966
C08179=1139.148,391.445,-86.828,-176.174,10.014,148.967
C08180=1139.144,391.692,-86.865,-176.174,10.016,148.967
C08181=1139.140,391.940,-86.902,-176.175,10.018,148.968
C08182=1139.137,392.187,-86.940,-176.176,10.021,148.969
C08183=1139.133,392.434,-86.977,-176.176,10.023,148.970
C08184=1139.129,392.681,-87.014,-176.177,10.025,148.970
C08185=1139.125,392.929,-87.052,-176.177,10.027,148.971
C08186=1139.122,393.175,-87.089,-176.178,10.029,148.972
C08187=1139.117,393.422,-87.126,-176.180,10.032,148.973
C08188=1139.114,393.670,-87.164,-176.181,10.034,148.974
C08189=1139.110,393.917,-87.201,-176.181,10.035,148.974
C08190=1139.107,394.164,-87.239,-176.182,10.038,148.975
C08191=1139.103,394.411,-87.276,-176.183,10.040,148.976
C08192=1139.098,394.659,-87.313,-176.184,10.042,148.977
C08193=1139.095,394.906,-87.351,-176.185,10.044,148.978
C08194=1139.091,395.153,-87.388,-176.186,10.046,148.978
C08195=1139.087,395.400,-87.425,-176.187,10.048,148.979
C08196=1139.084,395.648,-87.463,-176.188,10.050,148.980
C08197=1139.080,395.894,-87.500,-176.189,10.052,148.981
C08198=1139.076,396.141,-87.537,-176.190,10.054,148.982
C08199=1139.072,396.389,-87.575,-176.191,10.056,148.982
C08200=1139.068,396.636,-87.612,-176.192,10.059,148.983
C08201=1139.065,396.882,-87.649,-176.193,10.061,148.984
C08202=1139.061,397.130,-87.687,-176.194,10.063,148.985
C08203=1139.057,397.377,-87.724,-176.195,10.065,148.986
C08204=1139.053,397.624,-87.761,-176.197,10.067,148.987
C08205=1139.050,397.871,-87.799,-176.198,10.069,148.987
C08206=1139.046,398.119,-87.836,-176.199,10.071,148.988
C08207=1139.043,398.366,-87.874,-176.200,10.073,148.989
C08208=1139.039,398.613,-87.911,-176.201,10.075,148.990
C08209=1139.035,398.860,-87.948,-176.202,10.077,148.991
C08210=1139.031,399.108,-87.986,-176.203,10.079,148.992
C08211=1139.027,399.355,-88.022,-176.205,10.082,148.993
C08212=1139.023,399.601,-88.060,-176.206,10.084,148.993
C08213=1139.019,399.849,-88.098,-176.207,10.085,148.994
C08214=1139.015,400.096,-88.135,-176.208,10.087,148.995
C08215=1139.011,400.343,-88.172,-176.209,10.089,148.996
C08216=1139.008,400.591,-88.210,-176.211,10.091,148.997
C08217=1139.004,400.838,-88.247,-176.212,10.093,148.998
C08218=1139.000,401.084,-88.285,-176.213,10.095,148.999
C08219=1138.997,401.332,-88.322,-176.214,10.098,148.999
C08220=1138.993,401.579,-88.359,-176.215,10.100,149.000
C08221=1138.990,401.827,-88.397,-176.217,10.101,149.001
C08222=1138.986,402.073,-88.434,-176.218,10.103,149.002
C08223=1138.982,402.320,-88.471,-176.220,10.105,149.003
C08224=1138.978,402.568,-88.508,-176.221,10.107,149.004
C08225=1138.974,402.815,-88.546,-176.222,10.109,149.004
C08226=1138.970,403.062,-88.583,-176.223,10.112,149.005
C08227=1138.967,403.309,-88.621,-176.224,10.114,149.006
C08228=1138.963,403.556,-88.657,-176.225,10.116,149.007
C08229=1138.959,403.803,-88.695,-176.227,10.117,149.008
C08230=1138.956,404.051,-88.732,-176.228,10.119,149.009
C08231=1138.952,404.298,-88.770,-176.230,10.122,149.010
C08232=1138.948,404.545,-88.807,-176.231,10.124,149.011
C08233=1138.945,404.792,-88.845,-176.232,10.126,149.011
C08234=1138.940,405.039,-88.882,-176.233,10.128,149.012
C08235=1138.937,405.287,-88.920,-176.234,10.130,149.013
C08236=1138.933,405.534,-88.957,-176.235,10.132,149.014
C08237=1138.929,405.781,-88.994,-176.236,10.134,149.015
C08238=1138.925,406.028,-89.032,-176.238,10.136,149.016
C08239=1138.921,406.276,-89.069,-176.239,10.138,149.017
C08240=1138.917,406.522,-89.106,-176.240,10.140,149.017
C08241=1138.914,406.770,-89.143,-176.242,10.142,149.018
C08242=1138.910,407.017,-89.181,-176.243,10.144,149.019
C08243=1138.906,407.264,-89.218,-176.244,10.146,149.020
C08244=1138.903,407.511,-89.256,-176.245,10.148,149.021
C08245=1138.899,407.758,-89.293,-176.246,10.150,149.022
C08246=1138.895,408.005,-89.330,-176.247,10.152,149.023
C08247=1138.891,408.253,-89.367,-176.249,10.155,149.024
C08248=1138.888,408.499,-89.405,-176.250,10.157,149.024
C08249=1138.884,408.747,-89.442,-176.251,10.159,149.025
C08250=1138.880,408.994,-89.480,-176.252,10.161,149.026
C08251=1138.876,409.241,-89.517,-176.253,10.163,149.027
C08252=1138.873,409.488,-89.555,-176.254,10.165,149.028
C08253=1138.869,409.735,-89.591,-176.255,10.168,149.029
C08254=1138.865,409.982,-89.629,-176.256,10.170,149.029
C08255=1138.861,410.230,-89.667,-176.257,10.172,149.030
C08256=1138.857,410.477,-89.704,-176.258,10.175,149.031
C08257=1138.853,410.724,-89.741,-176.259,10.177,149.032
C08258=1138.850,410.972,-89.778,-176.260,10.179,149.033
C08259=1138.846,411.218,-89.816,-176.261,10.181,149.034
C08260=1138.842,411.466,-89.853,-176.262,10.183,149.035
C08261=1138.839,411.713,-89.891,-176.264,10.185,149.035
C08262=1138.834,411.960,-89.928,-176.265,10.187,149.036
C08263=1138.831,412.207,-89.966,-176.265,10.190,149.037
C08264=1138.827,412.455,-90.002,-176.266,10.192,149.038
C08265=1138.823,412.701,-90.040,-176.267,10.194,149.039
C08266=1138.820,412.949,-90.077,-176.268,10.196,149.040
C08267=1138.816,413.196,-90.115,-176.269,10.198,149.040
C08268=1138.812,413.443,-90.152,-176.270,10.201,149.041
C08269=1138.809,413.690,-90.190,-176.271,10.203,149.042
C08270=1138.805,413.937,-90.227,-176.272,10.205,149.043
C08271=1138.801,414.184,-90.264,-176.273,10.207,149.044
C08272=1138.797,414.432,-90.302,-176.274,10.209,149.044
C08273=1138.794,414.679,-90.339,-176.274,10.212,149.045
C08274=1138.791,414.927,-90.376,-176.275,10.214,149.046
C08275=1138.789,415.174,-90.413,-176.276,10.216,149.047
C08276=1138.788,415.421,-90.450,-176.277,10.218,149.048
C08277=1138.788,415.667,-90.488,-176.277,10.221,149.048
C08278=1138.788,415.915,-90.524,-176.278,10.223,149.049
C08279=1138.789,416.161,-90.561,-176.280,10.225,149.050
C08280=1138.790,416.451,-90.604,-176.281,10.227,149.051
C08281=1138.793,416.740,-90.647,-176.281,10.230,149.052
C08282=1138.797,417.029,-90.690,-176.282,10.232,149.053
C08283=1138.801,417.317,-90.733,-176.283,10.235,149.053
C08284=1138.382,417.317,-90.795,-176.986,11.602,149.592
C08285=1138.377,417.011,-90.750,-176.983,11.597,149.589
C08286=1138.373,416.705,-90.704,-176.979,11.592,149.587
C08287=1138.371,416.400,-90.658,-176.976,11.587,149.585
C08288=1138.369,416.094,-90.613,-176.973,11.582,149.583
C08289=1138.369,415.847,-90.575,-176.971,11.578,149.581
C08290=1138.368,415.599,-90.539,-176.968,11.574,149.580
C08291=1138.369,415.352,-90.501,-176.967,11.570,149.578
C08292=1138.370,415.105,-90.464,-176.964,11.566,149.576
C08293=1138.373,414.858,-90.426,-176.962,11.562,149.575
C08294=1138.375,414.611,-90.389,-176.959,11.558,149.573
C08295=1138.379,414.363,-90.352,-176.957,11.554,149.572
C08296=1138.382,414.117,-90.314,-176.955,11.550,149.570
C08297=1138.386,413.870,-90.276,-176.953,11.546,149.569
C08298=1138.389,413.623,-90.239,-176.951,11.542,149.567
C08299=1138.393,413.375,-90.200,-176.949,11.539,149.566
C08300=1138.397,413.128,-90.163,-176.947,11.534,149.564
C08301=1138.401,412.881,-90.125,-176.944,11.531,149.563
C08302=1138.404,412.634,-90.088,-176.943,11.527,149.561
C08303=1138.408,412.387,-90.050,-176.940,11.524,149.560
C08304=1138.412,412.140,-90.012,-176.939,11.520,149.558
C08305=1138.416,411.892,-89.974,-176.937,11.517,149.557
C08306=1138.419,411.646,-89.937,-176.935,11.512,149.555
C08307=1138.423,411.399,-89.899,-176.933,11.509,149.554
C08308=1138.427,411.151,-89.861,-176.931,11.505,149.553
C08309=1138.431,410.904,-89.824,-176.929,11.502,149.551
C08310=1138.434,410.657,-89.786,-176.928,11.498,149.550
C08311=1138.438,410.411,-89.748,-176.926,11.495,149.549
C08312=1138.442,410.163,-89.711,-176.924,11.491,149.547
C08313=1138.446,409.916,-89.673,-176.922,11.488,149.546
C08314=1138.449,409.669,-89.635,-176.921,11.485,149.545
C08315=1138.453,409.422,-89.597,-176.919,11.482,149.543
C08316=1138.457,409.174,-89.560,-176.918,11.478,149.542
C08317=1138.460,408.928,-89.523,-176.916,11.475,149.541
C08318=1138.464,408.680,-89.484,-176.915,11.472,149.540
C08319=1138.468,408.433,-89.446,-176.912,11.468,149.538
C08320=1138.472,408.186,-89.409,-176.911,11.465,149.537
C08321=1138.475,407.939,-89.372,-176.910,11.462,149.536
C08322=1138.479,407.692,-89.334,-176.908,11.459,149.535
C08323=1138.483,407.445,-89.296,-176.907,11.456,149.534
C08324=1138.487,407.198,-89.259,-176.905,11.453,149.532
C08325=1138.490,406.950,-89.221,-176.904,11.449,149.531
C08326=1138.494,406.704,-89.183,-176.902,11.447,149.530
C08327=1138.498,406.456,-89.145,-176.901,11.443,149.529
C08328=1138.502,406.209,-89.108,-176.900,11.441,149.528
C08329=1138.505,405.962,-89.070,-176.899,11.437,149.527
C08330=1138.509,405.715,-89.032,-176.897,11.435,149.526
C08331=1138.512,405.468,-88.994,-176.896,11.432,149.525
C08332=1138.517,405.220,-88.957,-176.895,11.429,149.524
C08333=1138.536,404.020,-88.778,-176.229,10.130,149.012
C08334=1138.539,403.779,-88.742,-176.228,10.128,149.011
C08335=1138.543,403.539,-88.705,-176.227,10.126,149.010
C08336=1138.546,403.298,-88.668,-176.226,10.124,149.009
C08337=1138.550,403.050,-88.632,-176.224,10.122,149.008
C08338=1138.553,402.803,-88.594,-176.223,10.120,149.008
C08339=1138.557,402.556,-88.557,-176.222,10.118,149.007
C08340=1138.561,402.309,-88.519,-176.220,10.116,149.006
C08341=1138.565,402.062,-88.482,-176.219,10.114,149.005
C08342=1138.568,401.815,-88.444,-176.218,10.112,149.004
C08343=1138.573,401.568,-88.408,-176.217,10.110,149.003
C08344=1138.576,401.321,-88.370,-176.216,10.108,149.002
C08345=1138.580,401.073,-88.333,-176.214,10.105,149.001
C08346=1138.584,400.826,-88.295,-176.213,10.103,149.001
C08347=1138.588,400.579,-88.257,-176.212,10.102,149.000
C08348=1138.592,400.332,-88.220,-176.211,10.100,148.999
C08349=1138.595,400.084,-88.183,-176.210,10.098,148.998
C08350=1138.599,399.838,-88.145,-176.208,10.095,148.997
C08351=1138.603,399.590,-88.108,-176.207,10.093,148.996
C08352=1138.606,399.343,-88.070,-176.206,10.091,148.995
C08353=1138.610,399.096,-88.033,-176.205,10.089,148.995
C08354=1138.614,398.849,-87.996,-176.204,10.087,148.994
C08355=1138.618,398.601,-87.959,-176.203,10.085,148.993
C08356=1138.621,398.355,-87.921,-176.202,10.083,148.992
C08357=1138.625,398.108,-87.884,-176.200,10.082,148.991
C08358=1138.629,397.860,-87.847,-176.199,10.080,148.991
C08359=1138.633,397.613,-87.809,-176.198,10.078,148.990
C08360=1138.636,397.365,-87.772,-176.196,10.075,148.989
C08361=1138.640,397.119,-87.735,-176.195,10.073,148.988
C08362=1138.644,396.872,-87.698,-176.194,10.071,148.987
C08363=1138.648,396.624,-87.659,-176.193,10.069,148.986
C08364=1138.652,396.377,-87.622,-176.192,10.067,148.985
C08365=1138.656,396.130,-87.585,-176.191,10.065,148.985
C08366=1138.659,395.882,-87.547,-176.190,10.063,148.984
C08367=1138.663,395.636,-87.510,-176.189,10.061,148.983
C08368=1138.667,395.389,-87.473,-176.188,10.059,148.982
C08369=1138.671,395.141,-87.435,-176.187,10.057,148.981
C08370=1138.675,394.894,-87.398,-176.186,10.054,148.981
C08371=1138.678,394.647,-87.360,-176.185,10.052,148.980
C08372=1138.682,394.400,-87.323,-176.184,10.050,148.979
C08373=1138.686,394.153,-87.286,-176.184,10.048,148.978
C08374=1138.689,393.905,-87.249,-176.182,10.046,148.977
C08375=1138.693,393.659,-87.211,-176.181,10.044,148.977
C08376=1138.697,393.411,-87.174,-176.181,10.041,148.976
C08377=1138.700,393.164,-87.136,-176.180,10.040,148.975
C08378=1138.704,392.917,-87.099,-176.179,10.037,148.974
C08379=1138.708,392.670,-87.062,-176.178,10.035,148.973
C08380=1138.712,392.422,-87.025,-176.178,10.033,148.973
C08381=1138.716,392.175,-86.988,-176.177,10.031,148.972
C08382=1138.719,391.928,-86.950,-176.177,10.028,148.971
C08383=1138.724,391.681,-86.912,-176.176,10.026,148.970
C08384=1138.728,391.434,-86.875,-176.175,10.024,148.970
C08385=1138.731,391.146,-86.832,-176.175,10.022,148.969
C08386=1138.736,390.859,-86.788,-176.174,10.019,148.968
C08387=1138.740,390.571,-86.745,-176.174,10.016,148.967
C08388=1138.745,390.284,-86.701,-176.173,10.013,148.966
C08389=1138.748,390.037,-86.664,-176.172,10.011,148.966
C08390=1138.753,389.790,-86.627,-176.172,10.008,148.965
C08391=1138.756,389.543,-86.589,-176.172,10.006,148.964
C08392=1138.760,389.295,-86.552,-176.171,10.004,148.963
C08393=1138.763,389.048,-86.514,-176.171,10.001,148.963
C08394=1138.767,388.801,-86.477,-176.171,9.999,148.962
C08395=1138.771,388.554,-86.441,-176.171,9.996,148.961
C08396=1138.774,388.307,-86.403,-176.171,9.994,148.961
C08397=1138.779,388.059,-86.366,-176.171,9.991,148.960
C08398=1138.782,387.813,-86.328,-176.171,9.989,148.959
C08399=1138.786,387.565,-86.291,-176.171,9.986,148.958
C08400=1138.790,387.318,-86.254,-176.170,9.984,148.958
C08401=1138.794,387.071,-86.216,-176.171,9.981,148.957
C08402=1138.797,386.823,-86.179,-176.171,9.978,148.956
C08403=1138.801,386.577,-86.142,-176.171,9.975,148.956
C08404=1138.805,386.329,-86.105,-176.171,9.973,148.955
C08405=1138.809,386.082,-86.068,-176.172,9.970,148.955
C08406=1138.812,385.835,-86.030,-176.172,9.967,148.954
C08407=1138.816,385.588,-85.993,-176.173,9.964,148.953
C08408=1138.820,385.340,-85.956,-176.173,9.962,148.953
C08409=1138.824,385.093,-85.918,-176.174,9.958,148.952
C08410=1138.828,384.846,-85.882,-176.175,9.955,148.951
C08411=1138.830,384.599,-85.844,-176.175,9.952,148.951
C08412=1138.834,384.352,-85.807,-176.176,9.950,148.950
C08413=1138.838,384.105,-85.770,-176.177,9.947,148.950
C08414=1138.843,383.858,-85.734,-176.177,9.944,148.949
C08415=1138.846,383.610,-85.696,-176.179,9.940,148.949
C08416=1138.850,383.363,-85.659,-176.180,9.937,148.948
C08417=1138.854,383.116,-85.622,-176.181,9.934,148.947
C08418=1138.857,382.869,-85.584,-176.182,9.931,148.947
C08419=1138.861,382.622,-85.547,-176.183,9.927,148.946
C08420=1138.865,382.374,-85.510,-176.185,9.924,148.946
C08421=1138.869,382.126,-85.473,-176.186,9.920,148.945
C08422=1138.873,381.880,-85.435,-176.187,9.917,148.945
C08423=1138.877,381.633,-85.399,-176.189,9.913,148.944
C08424=1138.880,381.386,-85.362,-176.190,9.910,148.944
C08425=1138.884,381.138,-85.325,-176.191,9.907,148.943
C08426=1138.888,380.891,-85.288,-176.193,9.903,148.943
C08427=1138.891,380.644,-85.251,-176.195,9.899,148.942
C08428=1138.895,380.397,-85.214,-176.197,9.896,148.942
C08429=1138.899,380.149,-85.177,-176.198,9.892,148.941
C08430=1138.903,379.902,-85.140,-176.200,9.889,148.941
C08431=1138.906,379.655,-85.104,-176.202,9.885,148.940
C08432=1138.911,379.408,-85.067,-176.204,9.881,148.940
C08433=1138.914,379.160,-85.029,-176.206,9.877,148.939
C08434=1138.918,378.913,-84.993,-176.208,9.874,148.939
C08435=1138.922,378.666,-84.955,-176.210,9.870,148.938
C08436=1138.926,378.419,-84.918,-176.211,9.866,148.938
C08437=1138.929,378.172,-84.882,-176.213,9.863,148.937
C08438=1138.933,377.924,-84.845,-176.215,9.858,148.937
C08439=1138.937,377.677,-84.808,-176.217,9.855,148.937
C08440=1138.941,377.430,-84.771,-176.220,9.850,148.936
C08441=1138.944,377.183,-84.735,-176.222,9.847,148.936
C08442=1138.948,376.936,-84.698,-176.224,9.843,148.935
C08443=1138.952,376.688,-84.661,-176.226,9.839,148.935
C08444=1138.956,376.441,-84.624,-176.228,9.835,148.934
C08445=1138.959,376.194,-84.587,-176.231,9.831,148.934
C08446=1138.964,375.946,-84.551,-176.233,9.826,148.933
C08447=1138.968,375.699,-84.514,-176.235,9.823,148.933
C08448=1138.972,375.452,-84.478,-176.238,9.818,148.933
C08449=1138.975,375.204,-84.441,-176.240,9.815,148.932
C08450=1138.979,374.957,-84.404,-176.242,9.811,148.932
C08451=1138.983,374.710,-84.367,-176.245,9.806,148.931
C08452=1138.986,374.463,-84.331,-176.247,9.802,148.931
C08453=1138.990,374.216,-84.294,-176.249,9.798,148.930
C08454=1138.995,373.968,-84.258,-176.252,9.794,148.930
C08455=1138.998,373.721,-84.222,-176.254,9.789,148.929
C08456=1139.002,373.474,-84.185,-176.257,9.785,148.929
C08457=1139.005,373.226,-84.148,-176.260,9.781,148.929
C08458=1139.009,372.978,-84.112,-176.262,9.777,148.928
C08459=1139.014,372.731,-84.075,-176.264,9.773,148.928
C08460=1139.017,372.484,-84.039,-176.267,9.769,148.927
C08461=1139.021,372.237,-84.002,-176.269,9.764,148.927
C08462=1139.025,371.990,-83.967,-176.272,9.760,148.927
C08463=1139.029,371.742,-83.930,-176.275,9.756,148.926
C08464=1139.032,371.495,-83.893,-176.277,9.751,148.926
C08465=1139.036,371.248,-83.857,-176.280,9.747,148.925
C08466=1139.041,371.000,-83.820,-176.282,9.743,148.925
C08467=1139.044,370.753,-83.785,-176.285,9.739,148.924
C08468=1139.048,370.506,-83.748,-176.288,9.734,148.924
C08469=1139.052,370.259,-83.712,-176.290,9.731,148.924
C08470=1139.056,370.011,-83.676,-176.292,9.726,148.923
C08471=1139.059,369.763,-83.639,-176.295,9.722,148.923
C08472=1139.063,369.516,-83.603,-176.298,9.718,148.922
C08473=1139.067,369.269,-83.567,-176.300,9.713,148.922
C08474=1139.070,369.021,-83.531,-176.303,9.709,148.922
C08475=1139.074,368.774,-83.494,-176.306,9.705,148.921
C08476=1139.078,368.527,-83.459,-176.308,9.701,148.921
C08477=1139.082,368.279,-83.422,-176.311,9.696,148.920
C08478=1139.086,368.032,-83.386,-176.314,9.692,148.920
C08479=1139.090,367.784,-83.350,-176.316,9.688,148.920
C08480=1139.094,367.538,-83.314,-176.319,9.683,148.919
C08481=1139.098,367.290,-83.279,-176.321,9.679,148.919
C08482=1139.102,367.043,-83.242,-176.324,9.675,148.918
C08483=1139.106,366.796,-83.206,-176.327,9.671,148.918
C08484=1139.110,366.548,-83.170,-176.329,9.666,148.917
C08485=1139.113,366.301,-83.134,-176.332,9.662,148.917
C08486=1139.117,366.054,-83.098,-176.335,9.658,148.917
C08487=1139.121,365.806,-83.062,-176.337,9.653,148.916
C08488=1139.125,365.558,-83.027,-176.340,9.649,148.916
C08489=1139.129,365.275,-82.986,-176.343,9.644,148.915
C08490=1139.134,364.990,-82.944,-176.346,9.639,148.915
C08491=1139.138,364.707,-82.903,-176.349,9.635,148.914
C08492=1139.142,364.423,-82.862,-176.352,9.629,148.914
C08493=1139.147,364.175,-82.826,-176.355,9.625,148.914
C08494=1139.150,363.928,-82.790,-176.357,9.621,148.913
C08495=1139.154,363.681,-82.754,-176.360,9.617,148.913
C08496=1139.157,363.433,-82.719,-176.363,9.612,148.912
C08497=1139.162,363.186,-82.683,-176.365,9.608,148.912
C08498=1139.166,362.939,-82.647,-176.368,9.604,148.912
C08499=1139.170,362.691,-82.612,-176.370,9.599,148.911
C08500=1139.173,362.444,-82.576,-176.373,9.595,148.911
C08501=1139.177,362.196,-82.541,-176.376,9.591,148.910
C08502=1139.181,361.949,-82.505,-176.378,9.587,148.910
C08503=1139.185,361.701,-82.469,-176.381,9.583,148.910
C08504=1139.189,361.454,-82.434,-176.383,9.579,148.909
C08505=1139.193,361.207,-82.398,-176.386,9.574,148.909
C08506=1139.197,360.959,-82.363,-176.389,9.570,148.909
C08507=1139.200,360.712,-82.327,-176.391,9.566,148.908
C08508=1139.204,360.464,-82.292,-176.394,9.562,148.908
C08509=1139.208,360.217,-82.256,-176.396,9.557,148.907
C08510=1139.212,359.970,-82.221,-176.398,9.554,148.907
C08511=1139.216,359.722,-82.185,-176.401,9.550,148.907
C08512=1139.220,359.474,-82.149,-176.403,9.545,148.906
C08513=1139.224,359.227,-82.114,-176.406,9.541,148.906
C08514=1139.228,358.980,-82.078,-176.409,9.537,148.905
C08515=1139.232,358.732,-82.044,-176.411,9.533,148.905
C08516=1139.236,358.485,-82.008,-176.414,9.529,148.905
C08517=1139.239,358.237,-81.973,-176.416,9.525,148.904
C08518=1139.243,357.990,-81.937,-176.419,9.520,148.904
C08519=1139.247,357.743,-81.902,-176.422,9.516,148.904
C08520=1139.251,357.495,-81.867,-176.424,9.513,148.903
C08521=1139.255,357.247,-81.831,-176.426,9.508,148.903
C08522=1139.259,357.000,-81.796,-176.429,9.504,148.902
C08523=1139.263,356.753,-81.761,-176.432,9.500,148.902
C08524=1139.267,356.505,-81.726,-176.434,9.496,148.902
C08525=1139.270,356.257,-81.690,-176.436,9.492,148.901
C08526=1139.275,356.010,-81.655,-176.439,9.488,148.901
C08527=1139.279,355.762,-81.620,-176.441,9.483,148.900
C08528=1139.282,355.515,-81.585,-176.444,9.480,148.900
C08529=1139.286,355.268,-81.550,-176.446,9.476,148.900
C08530=1139.290,355.020,-81.515,-176.449,9.471,148.899
C08531=1139.293,354.773,-81.480,-176.452,9.467,148.899
C08532=1139.298,354.525,-81.445,-176.454,9.464,148.899
C08533=1139.302,354.278,-81.410,-176.457,9.460,148.898
C08534=1139.306,354.030,-81.375,-176.459,9.455,148.898
C08535=1139.310,353.783,-81.340,-176.462,9.451,148.897
C08536=1139.313,353.535,-81.304,-176.464,9.448,148.897
C08537=1139.317,353.287,-81.269,-176.466,9.443,148.897
C08538=1139.322,353.040,-81.235,-176.469,9.439,148.896
C08539=1139.325,352.793,-81.200,-176.472,9.435,148.896
C08540=1139.329,352.544,-81.165,-176.474,9.431,148.896
C08541=1139.333,352.298,-81.130,-176.477,9.427,148.895
C08542=1139.337,352.050,-81.095,-176.479,9.423,148.895
C08543=1139.341,351.803,-81.060,-176.482,9.419,148.895
C08544=1139.345,351.555,-81.026,-176.484,9.415,148.894
C08545=1139.349,351.307,-80.991,-176.487,9.411,148.894
C08546=1139.353,351.060,-80.956,-176.490,9.407,148.894
C08547=1139.357,350.812,-80.921,-176.492,9.403,148.893
C08548=1139.361,350.565,-80.886,-176.494,9.399,148.893
C08549=1139.364,350.317,-80.851,-176.497,9.395,148.892
C08550=1139.369,350.070,-80.817,-176.500,9.391,148.892
C08551=1139.373,349.822,-80.782,-176.502,9.387,148.892
C08552=1139.377,349.574,-80.747,-176.504,9.383,148.891
C08553=1139.380,349.327,-80.713,-176.507,9.379,148.891
C08554=1139.384,349.079,-80.678,-176.509,9.375,148.891
C08555=1139.389,348.832,-80.643,-176.512,9.371,148.890
C08556=1139.392,348.584,-80.608,-176.515,9.367,148.890
C08557=1139.396,348.337,-80.574,-176.517,9.363,148.890
C08558=1139.400,348.089,-80.539,-176.519,9.359,148.889
C08559=1139.404,347.842,-80.505,-176.522,9.355,148.889
C08560=1139.408,347.594,-80.470,-176.525,9.351,148.889
C08561=1139.413,347.346,-80.436,-176.527,9.347,148.888
C08562=1139.416,347.099,-80.401,-176.530,9.343,148.888
C08563=1139.420,346.852,-80.367,-176.533,9.339,148.888
C08564=1139.424,346.604,-80.332,-176.535,9.335,148.887
C08565=1139.428,346.356,-80.298,-176.538,9.331,148.887
C08566=1139.432,346.108,-80.263,-176.540,9.327,148.887
C08567=1139.436,345.861,-80.229,-176.542,9.324,148.886
C08568=1139.440,345.613,-80.194,-176.545,9.319,148.886
C08569=1139.444,345.366,-80.160,-176.548,9.315,148.886
C08570=1139.448,345.119,-80.126,-176.550,9.311,148.885
C08571=1139.452,344.870,-80.091,-176.553,9.307,148.885
C08572=1139.456,344.623,-80.057,-176.555,9.303,148.885
C08573=1139.460,344.375,-80.022,-176.558,9.300,148.884
C08574=1139.464,344.128,-79.989,-176.560,9.296,148.884
C08575=1139.468,343.880,-79.954,-176.563,9.291,148.884
C08576=1139.472,343.633,-79.920,-176.565,9.288,148.884
C08577=1139.476,343.385,-79.885,-176.568,9.284,148.883
C08578=1139.480,343.137,-79.852,-176.571,9.280,148.883
C08579=1139.484,342.890,-79.817,-176.573,9.276,148.882
C08580=1139.488,342.642,-79.783,-176.576,9.272,148.882
C08581=1139.492,342.394,-79.749,-176.578,9.268,148.882
C08582=1139.496,342.147,-79.715,-176.580,9.264,148.882
C08583=1139.500,341.899,-79.680,-176.583,9.260,148.881
C08584=1139.504,341.651,-79.647,-176.586,9.256,148.881
C08585=1139.508,341.404,-79.613,-176.588,9.253,148.881
C08586=1139.512,341.156,-79.578,-176.591,9.248,148.880
C08587=1139.516,340.909,-79.544,-176.594,9.244,148.880
C08588=1139.521,340.661,-79.511,-176.596,9.241,148.880
C08589=1139.524,340.413,-79.476,-176.598,9.236,148.879
C08590=1139.528,340.166,-79.442,-176.601,9.232,148.879
C08591=1139.532,339.918,-79.409,-176.604,9.229,148.879
C08592=1139.536,339.670,-79.374,-176.606,9.225,148.878
C08593=1139.540,339.390,-79.336,-176.609,9.221,148.878
C08594=1139.545,339.109,-79.297,-176.612,9.216,148.878
C08595=1139.550,338.828,-79.259,-176.615,9.211,148.878
C08596=1139.555,338.548,-79.220,-176.618,9.207,148.877
C08597=1139.558,338.300,-79.186,-176.620,9.204,148.877
C08598=1139.562,338.052,-79.153,-176.623,9.200,148.877
C08599=1139.567,337.805,-79.119,-176.626,9.196,148.876
C08600=1139.571,337.557,-79.085,-176.628,9.192,148.876
C08601=1139.574,337.309,-79.051,-176.631,9.188,148.876
C08602=1139.578,337.062,-79.018,-176.634,9.184,148.876
C08603=1139.583,336.814,-78.984,-176.636,9.180,148.875
C08604=1139.586,336.566,-78.950,-176.639,9.176,148.875
C08605=1139.590,336.319,-78.916,-176.641,9.173,148.875
C08606=1139.594,336.071,-78.883,-176.643,9.169,148.874
C08607=1139.598,335.824,-78.849,-176.646,9.165,148.874
C08608=1139.602,335.575,-78.815,-176.649,9.161,148.874
C08609=1139.606,335.328,-78.781,-176.651,9.157,148.873
C08610=1139.610,335.080,-78.748,-176.653,9.154,148.873
C08611=1139.614,334.832,-78.715,-176.656,9.150,148.873
C08612=1139.618,334.585,-78.681,-176.659,9.145,148.873
C08613=1139.622,334.337,-78.647,-176.661,9.142,148.872
C08614=1139.627,334.089,-78.614,-176.664,9.138,148.872
C08615=1139.630,333.842,-78.580,-176.667,9.135,148.872
C08616=1139.635,333.594,-78.547,-176.669,9.130,148.871
C08617=1139.639,333.346,-78.514,-176.672,9.126,148.871
C08618=1139.642,333.098,-78.479,-176.674,9.123,148.871
C08619=1139.646,332.851,-78.446,-176.677,9.119,148.871
C08620=1139.650,332.603,-78.413,-176.679,9.115,148.870
C08621=1139.654,332.355,-78.380,-176.682,9.111,148.870
C08622=1139.658,332.108,-78.346,-176.685,9.107,148.870
C08623=1139.662,331.860,-78.313,-176.687,9.104,148.870
C08624=1139.667,331.612,-78.279,-176.690,9.099,148.869
C08625=1139.671,331.364,-78.246,-176.692,9.096,148.869
C08626=1139.675,331.116,-78.212,-176.695,9.092,148.869
C08627=1139.679,330.869,-78.179,-176.697,9.089,148.869
C08628=1139.683,330.621,-78.145,-176.700,9.085,148.868
C08629=1139.687,330.374,-78.112,-176.703,9.080,148.868
C08630=1139.691,330.126,-78.079,-176.705,9.077,148.868
C08631=1139.695,329.878,-78.046,-176.708,9.073,148.868
C08632=1139.699,329.630,-78.012,-176.710,9.070,148.867
C08633=1139.703,329.382,-77.979,-176.713,9.066,148.867
C08634=1139.707,329.134,-77.946,-176.715,9.062,148.867
C08635=1139.711,328.887,-77.913,-176.718,9.058,148.866
C08636=1139.715,328.639,-77.880,-176.721,9.054,148.866
C08637=1139.719,328.391,-77.847,-176.724,9.051,148.866
C08638=1139.723,328.144,-77.814,-176.726,9.047,148.866
C08639=1139.727,327.896,-77.781,-176.729,9.043,148.866
C08640=1139.731,327.648,-77.748,-176.731,9.039,148.865
C08641=1139.735,327.401,-77.715,-176.734,9.036,148.865
C08642=1139.739,327.153,-77.681,-176.737,9.032,148.865
C08643=1139.744,326.905,-77.648,-176.739,9.028,148.865
C08644=1139.748,326.657,-77.615,-176.742,9.024,148.864
C08645=1139.752,326.409,-77.583,-176.744,9.021,148.864
C08646=1139.756,326.162,-77.550,-176.747,9.017,148.864
C08647=1139.760,325.914,-77.517,-176.750,9.013,148.863
C08648=1139.764,325.666,-77.484,-176.752,9.009,148.863
C08649=1139.768,325.418,-77.451,-176.755,9.005,148.863
C08650=1139.772,325.171,-77.417,-176.757,9.002,148.863
C08651=1139.777,324.922,-77.385,-176.760,8.998,148.863
C08652=1139.780,324.675,-77.352,-176.762,8.995,148.862
C08653=1139.784,324.427,-77.319,-176.765,8.991,148.862
C08654=1139.788,324.179,-77.286,-176.768,8.987,148.862
C08655=1139.793,323.931,-77.254,-176.771,8.983,148.862
C08656=1139.796,323.684,-77.221,-176.773,8.980,148.861
C08657=1139.800,323.436,-77.188,-176.776,8.976,148.861
C08658=1139.804,323.188,-77.155,-176.778,8.972,148.861
C08659=1139.809,322.940,-77.122,-176.781,8.968,148.861
C08660=1139.812,322.692,-77.090,-176.783,8.965,148.861
C08661=1139.816,322.445,-77.057,-176.786,8.961,148.860
C08662=1139.821,322.196,-77.024,-176.788,8.958,148.860
C08663=1139.824,321.949,-76.992,-176.791,8.954,148.860
C08664=1139.829,321.701,-76.959,-176.794,8.950,148.860
C08665=1139.833,321.453,-76.926,-176.797,8.946,148.859
C08666=1139.836,321.205,-76.894,-176.799,8.943,148.859
C08667=1139.841,320.957,-76.861,-176.802,8.939,148.859
C08668=1139.845,320.709,-76.828,-176.804,8.936,148.859
C08669=1139.849,320.462,-76.796,-176.807,8.932,148.859
C08670=1139.853,320.214,-76.763,-176.809,8.928,148.858
C08671=1139.857,319.966,-76.731,-176.812,8.924,148.858
C08672=1139.861,319.719,-76.698,-176.815,8.921,148.858
C08673=1139.866,319.470,-76.666,-176.818,8.917,148.858
C08674=1139.869,319.223,-76.633,-176.820,8.914,148.858
C08675=1139.873,318.974,-76.601,-176.823,8.910,148.857
C08676=1139.877,318.726,-76.569,-176.825,8.906,148.857
C08677=1139.882,318.479,-76.536,-176.828,8.902,148.857
C08678=1139.885,318.231,-76.504,-176.831,8.899,148.857
C08679=1139.890,317.984,-76.471,-176.833,8.895,148.857
C08680=1139.894,317.735,-76.439,-176.836,8.892,148.856
C08681=1139.898,317.487,-76.407,-176.839,8.888,148.856
C08682=1139.902,317.239,-76.374,-176.841,8.884,148.856
C08683=1139.906,316.991,-76.342,-176.844,8.880,148.856
C08684=1139.911,316.744,-76.310,-176.846,8.877,148.856
C08685=1139.914,316.496,-76.277,-176.849,8.873,148.855
C08686=1139.919,316.248,-76.245,-176.852,8.870,148.855
C08687=1139.922,316.000,-76.213,-176.855,8.866,148.855
C08688=1139.926,315.752,-76.181,-176.857,8.862,148.855
C08689=1139.931,315.505,-76.148,-176.860,8.858,148.855
C08690=1139.934,315.257,-76.117,-176.862,8.855,148.854
C08691=1139.939,315.009,-76.084,-176.865,8.852,148.854
C08692=1139.943,314.760,-76.052,-176.867,8.848,148.854
C08693=1139.948,314.513,-76.020,-176.870,8.844,148.854
C08694=1139.951,314.265,-75.988,-176.873,8.840,148.854
C08695=1139.955,314.017,-75.956,-176.875,8.837,148.853
C08696=1139.959,313.769,-75.923,-176.878,8.833,148.853
C08697=1139.963,313.492,-75.888,-176.881,8.829,148.853
C08698=1139.968,313.214,-75.852,-176.884,8.825,148.853
C08699=1139.973,312.936,-75.817,-176.887,8.821,148.853
C08700=1139.978,312.658,-75.780,-176.890,8.817,148.852
C08701=1139.982,312.410,-75.749,-176.892,8.814,148.852
C08702=1139.986,312.161,-75.716,-176.895,8.810,148.852
C08703=1139.990,311.913,-75.684,-176.898,8.807,148.852
C08704=1139.994,311.666,-75.653,-176.900,8.803,148.852
C08705=1139.999,311.418,-75.620,-176.903,8.799,148.851
C08706=1140.002,311.170,-75.589,-176.906,8.796,148.852
C08707=1140.007,310.922,-75.557,-176.909,8.792,148.851
C08708=1140.011,310.674,-75.525,-176.911,8.789,148.851
C08709=1140.015,310.426,-75.493,-176.914,8.785,148.851
C08710=1140.019,310.178,-75.461,-176.916,8.782,148.851
C08711=1140.023,309.930,-75.429,-176.919,8.778,148.851
C08712=1140.027,309.682,-75.398,-176.922,8.774,148.850
C08713=1140.032,309.435,-75.366,-176.924,8.771,148.850
C08714=1140.035,309.187,-75.334,-176.927,8.767,148.850
C08715=1140.039,308.938,-75.303,-176.930,8.764,148.850
C08716=1140.044,308.691,-75.271,-176.933,8.760,148.850
C08717=1140.048,308.442,-75.239,-176.935,8.757,148.850
C08718=1140.052,308.195,-75.207,-176.937,8.753,148.849
C08719=1140.056,307.947,-75.175,-176.941,8.750,148.849
C08720=1140.060,307.698,-75.144,-176.943,8.746,148.849
C08721=1140.065,307.451,-75.113,-176.946,8.742,148.849
C08722=1140.068,307.203,-75.081,-176.948,8.739,148.849
C08723=1140.073,306.955,-75.049,-176.951,8.736,148.849
C08724=1140.077,306.707,-75.018,-176.953,8.732,148.848
C08725=1140.081,306.459,-74.986,-176.956,8.729,148.848
C08726=1140.085,306.211,-74.954,-176.959,8.725,148.848
C08727=1140.089,305.963,-74.923,-176.962,8.721,148.848
C08728=1140.094,305.715,-74.892,-176.964,8.718,148.848
C08729=1140.097,305.467,-74.860,-176.967,8.714,148.848
C08730=1140.102,305.219,-74.829,-176.970,8.711,148.848
C08731=1140.106,304.971,-74.797,-176.972,8.707,148.847
C08732=1140.111,304.724,-74.765,-176.975,8.704,148.847
C08733=1140.115,304.475,-74.734,-176.977,8.701,148.847
C08734=1140.119,304.228,-74.703,-176.981,8.697,148.847
C08735=1140.123,303.979,-74.671,-176.983,8.694,148.847
C08736=1140.127,303.732,-74.640,-176.986,8.690,148.847
C08737=1140.131,303.483,-74.609,-176.988,8.686,148.847
C08738=1140.136,303.236,-74.577,-176.991,8.683,148.847
C08739=1140.140,302.987,-74.546,-176.994,8.679,148.846
C08740=1140.144,302.740,-74.515,-176.996,8.676,148.846
C08741=1140.148,302.491,-74.484,-176.999,8.673,148.846
C08742=1140.152,302.244,-74.452,-177.002,8.669,148.846
C08743=1140.156,301.995,-74.421,-177.004,8.666,148.846
C08744=1140.161,301.748,-74.390,-177.007,8.662,148.846
C08745=1140.165,301.499,-74.358,-177.010,8.659,148.846
C08746=1140.169,301.251,-74.328,-177.012,8.655,148.845
C08747=1140.173,301.003,-74.296,-177.015,8.651,148.845
C08748=1140.177,300.755,-74.266,-177.018,8.648,148.845
C08749=1140.181,300.507,-74.234,-177.020,8.645,148.845
C08750=1140.185,300.259,-74.203,-177.023,8.641,148.845
C08751=1140.190,300.011,-74.172,-177.026,8.638,148.845
C08752=1140.194,299.763,-74.141,-177.028,8.635,148.845
C08753=1140.198,299.515,-74.110,-177.031,8.631,148.845
C08754=1140.202,299.267,-74.079,-177.034,8.628,148.844
C08755=1140.207,299.019,-74.048,-177.036,8.625,148.844
C08756=1140.211,298.771,-74.018,-177.039,8.621,148.844
C08757=1140.214,298.523,-73.986,-177.042,8.617,148.844
C08758=1140.219,298.275,-73.955,-177.044,8.614,148.844
C08759=1140.223,298.026,-73.924,-177.047,8.610,148.844
C08760=1140.228,297.778,-73.893,-177.050,8.607,148.844
C08761=1140.232,297.531,-73.862,-177.053,8.603,148.844
C08762=1140.235,297.283,-73.831,-177.055,8.600,148.843
C08763=1140.240,297.035,-73.800,-177.058,8.597,148.843
C08764=1140.244,296.786,-73.769,-177.061,8.593,148.843
C08765=1140.248,296.538,-73.738,-177.063,8.590,148.843
C08766=1140.252,296.291,-73.708,-177.066,8.587,148.843
C08767=1140.256,296.042,-73.677,-177.069,8.583,148.843
C08768=1140.261,295.794,-73.646,-177.072,8.580,148.843
C08769=1140.265,295.546,-73.616,-177.074,8.576,148.843
C08770=1140.269,295.298,-73.585,-177.077,8.573,148.843
C08771=1140.273,295.050,-73.554,-177.080,8.569,148.842
C08772=1140.278,294.802,-73.523,-177.082,8.566,148.842
C08773=1140.281,294.554,-73.492,-177.085,8.563,148.842
C08774=1140.286,294.306,-73.461,-177.088,8.559,148.842
C08775=1140.290,294.058,-73.431,-177.090,8.556,148.842
C08776=1140.294,293.810,-73.401,-177.093,8.553,148.842
C08777=1140.298,293.561,-73.370,-177.096,8.549,148.842
C08778=1140.303,293.313,-73.339,-177.098,8.546,148.842
C08779=1140.307,293.066,-73.309,-177.101,8.543,148.842
C08780=1140.311,292.817,-73.278,-177.104,8.539,148.842
C08781=1140.315,292.569,-73.248,-177.107,8.536,148.841
C08782=1140.319,292.321,-73.217,-177.109,8.532,148.841
C08783=1140.324,292.073,-73.186,-177.112,8.529,148.841
C08784=1140.327,291.825,-73.156,-177.115,8.525,148.841
C08785=1140.332,291.577,-73.125,-177.117,8.522,148.841
C08786=1140.336,291.329,-73.096,-177.120,8.519,148.841
C08787=1140.341,291.081,-73.065,-177.123,8.515,148.841
C08788=1140.344,290.832,-73.034,-177.125,8.512,148.841
C08789=1140.349,290.584,-73.004,-177.128,8.509,148.841
C08790=1140.352,290.337,-72.973,-177.131,8.505,148.841
C08791=1140.357,290.088,-72.943,-177.133,8.502,148.841
C08792=1140.361,289.840,-72.913,-177.136,8.499,148.841
C08793=1140.365,289.592,-72.882,-177.139,8.496,148.840
C08794=1140.369,289.344,-72.853,-177.142,8.492,148.840
C08795=1140.374,289.096,-72.822,-177.144,8.489,148.840
C08796=1140.378,288.848,-72.792,-177.147,8.486,148.840
C08797=1140.383,288.599,-72.762,-177.150,8.482,148.840
C08798=1140.386,288.351,-72.731,-177.153,8.479,148.840
C08799=1140.391,288.103,-72.700,-177.155,8.476,148.840
C08800=1140.395,287.855,-72.671,-177.158,8.473,148.840
C08801=1140.400,287.579,-72.637,-177.161,8.469,148.840
C08802=1140.404,287.304,-72.603,-177.164,8.465,148.840
C08803=1140.409,287.028,-72.570,-177.167,8.461,148.840
C08804=1140.414,286.753,-72.536,-177.170,8.458,148.840
C08805=1140.418,286.505,-72.507,-177.173,8.454,148.839
C08806=1140.422,286.256,-72.476,-177.176,8.451,148.839
C08807=1140.426,286.008,-72.446,-177.178,8.447,148.839
C08808=1140.430,285.760,-72.416,-177.181,8.445,148.839
C08809=1140.435,285.512,-72.386,-177.184,8.440,148.839
C08810=1140.439,285.264,-72.356,-177.186,8.438,148.839
C08811=1140.443,285.016,-72.327,-177.189,8.434,148.839
C08812=1140.448,284.768,-72.296,-177.192,8.431,148.839
C08813=1140.452,284.520,-72.266,-177.194,8.427,148.839
C08814=1140.456,284.272,-72.236,-177.197,8.424,148.839
C08815=1140.461,284.023,-72.206,-177.200,8.421,148.839
C08816=1140.465,283.775,-72.177,-177.202,8.418,148.839
C08817=1140.468,283.527,-72.146,-177.205,8.414,148.839
C08818=1140.473,283.278,-72.116,-177.208,8.411,148.839
C08819=1140.477,283.031,-72.086,-177.211,8.408,148.839
C08820=1140.481,282.782,-72.056,-177.213,8.405,148.839
C08821=1140.485,282.534,-72.027,-177.217,8.401,148.839
C08822=1140.490,282.285,-71.997,-177.219,8.398,148.838
C08823=1140.494,282.038,-71.967,-177.222,8.395,148.838
C08824=1140.498,281.790,-71.937,-177.224,8.392,148.838
C08825=1140.503,281.541,-71.908,-177.227,8.388,148.838
C08826=1140.506,281.294,-71.878,-177.230,8.385,148.838
C08827=1140.511,281.045,-71.848,-177.233,8.382,148.838
C08828=1140.516,280.797,-71.818,-177.235,8.379,148.838
C08829=1140.520,280.548,-71.789,-177.238,8.375,148.838
C08830=1140.524,280.300,-71.759,-177.241,8.372,148.838
C08831=1140.528,280.053,-71.729,-177.243,8.369,148.838
C08832=1140.533,279.804,-71.699,-177.246,8.366,148.838
C08833=1140.537,279.556,-71.670,-177.249,8.363,148.838
C08834=1140.541,279.307,-71.640,-177.252,8.359,148.838
C08835=1140.545,279.059,-71.611,-177.255,8.356,148.838
C08836=1140.549,278.811,-71.581,-177.257,8.353,148.838
C08837=1140.554,278.563,-71.552,-177.260,8.350,148.838
C08838=1140.558,278.314,-71.522,-177.263,8.347,148.838
C08839=1140.562,278.066,-71.493,-177.266,8.343,148.838
C08840=1140.567,277.819,-71.464,-177.268,8.340,148.838
C08841=1140.571,277.571,-71.434,-177.271,8.336,148.838
C08842=1140.575,277.323,-71.404,-177.273,8.334,148.838
C08843=1140.579,277.074,-71.375,-177.276,8.331,148.838
C08844=1140.583,276.826,-71.345,-177.279,8.327,148.837
C08845=1140.587,276.578,-71.316,-177.282,8.324,148.837
C08846=1140.593,276.329,-71.286,-177.284,8.320,148.837
C08847=1140.597,276.080,-71.257,-177.287,8.317,148.837
C08848=1140.601,275.832,-71.228,-177.290,8.315,148.837
C08849=1140.604,275.584,-71.199,-177.293,8.310,148.837
C08850=1140.609,275.336,-71.169,-177.296,8.308,148.837
C08851=1140.613,275.088,-71.140,-177.298,8.305,148.837
C08852=1140.618,274.840,-71.111,-177.301,8.301,148.837
C08853=1140.622,274.592,-71.081,-177.303,8.298,148.837
C08854=1140.626,274.344,-71.052,-177.307,8.295,148.837
C08855=1140.630,274.095,-71.022,-177.309,8.291,148.837
C08856=1140.635,273.846,-70.994,-177.312,8.288,148.837
C08857=1140.639,273.598,-70.964,-177.315,8.286,148.837
C08858=1140.643,273.350,-70.935,-177.317,8.282,148.837
C08859=1140.648,273.102,-70.906,-177.320,8.279,148.837
C08860=1140.652,272.854,-70.876,-177.323,8.276,148.837
C08861=1140.656,272.605,-70.847,-177.326,8.272,148.837
C08862=1140.661,272.357,-70.818,-177.328,8.269,148.837
C08863=1140.664,272.109,-70.789,-177.331,8.267,148.837
C08864=1140.669,271.861,-70.761,-177.334,8.263,148.837
C08865=1140.673,271.612,-70.731,-177.337,8.260,148.837
C08866=1140.677,271.364,-70.702,-177.340,8.257,148.837
C08867=1140.682,271.115,-70.673,-177.342,8.253,148.837
C08868=1140.686,270.867,-70.644,-177.345,8.250,148.837
C08869=1140.690,270.620,-70.615,-177.348,8.247,148.837
C08870=1140.695,270.371,-70.586,-177.350,8.245,148.837
C08871=1140.699,270.123,-70.557,-177.353,8.241,148.837
C08872=1140.703,269.874,-70.528,-177.356,8.238,148.837
C08873=1140.708,269.626,-70.499,-177.359,8.235,148.837
C08874=1140.712,269.378,-70.470,-177.361,8.231,148.837
C08875=1140.716,269.129,-70.442,-177.364,8.228,148.837
C08876=1140.720,268.881,-70.412,-177.367,8.226,148.837
C08877=1140.725,268.633,-70.384,-177.370,8.223,148.837
C08878=1140.729,268.385,-70.355,-177.373,8.219,148.837
C08879=1140.733,268.136,-70.326,-177.375,8.216,148.837
C08880=1140.737,267.888,-70.297,-177.378,8.213,148.837
C08881=1140.743,267.640,-70.268,-177.380,8.209,148.837
C08882=1140.746,267.392,-70.239,-177.383,8.207,148.837
C08883=1140.750,267.143,-70.211,-177.386,8.204,148.837
C08884=1140.755,266.895,-70.182,-177.389,8.201,148.837
C08885=1140.759,266.647,-70.153,-177.392,8.197,148.837
C08886=1140.763,266.398,-70.124,-177.395,8.194,148.837
C08887=1140.768,266.150,-70.096,-177.397,8.191,148.837
C08888=1140.772,265.902,-70.068,-177.400,8.188,148.837
C08889=1140.776,265.653,-70.038,-177.402,8.185,148.837
C08890=1140.781,265.405,-70.010,-177.405,8.182,148.837
C08891=1140.785,265.156,-69.982,-177.408,8.179,148.837
C08892=1140.789,264.908,-69.952,-177.411,8.176,148.837
C08893=1140.794,264.660,-69.924,-177.414,8.172,148.837
C08894=1140.798,264.411,-69.896,-177.417,8.169,148.837
C08895=1140.803,264.163,-69.867,-177.419,8.166,148.837
C08896=1140.807,263.915,-69.838,-177.422,8.163,148.837
C08897=1140.811,263.666,-69.810,-177.425,8.160,148.837
C08898=1140.815,263.419,-69.782,-177.427,8.157,148.837
C08899=1140.820,263.170,-69.753,-177.430,8.154,148.837
C08900=1140.823,262.922,-69.724,-177.433,8.151,148.837
C08901=1140.828,262.674,-69.696,-177.436,8.148,148.837
C08902=1140.832,262.425,-69.668,-177.439,8.144,148.837
C08903=1140.837,262.177,-69.639,-177.441,8.141,148.837
C08904=1140.841,261.928,-69.611,-177.444,8.138,148.837
C08905=1140.846,261.655,-69.579,-177.447,8.135,148.837
C08906=1140.850,261.381,-69.548,-177.450,8.131,148.837
C08907=1140.856,261.107,-69.517,-177.453,8.129,148.837
C08908=1140.860,260.834,-69.486,-177.456,8.125,148.837
C08909=1140.865,260.585,-69.457,-177.459,8.122,148.837
C08910=1140.869,260.337,-69.430,-177.462,8.119,148.837
C08911=1140.874,260.088,-69.401,-177.464,8.116,148.837
C08912=1140.878,259.841,-69.372,-177.467,8.113,148.837
C08913=1140.881,259.593,-69.344,-177.470,8.110,148.837
C08914=1140.886,259.344,-69.316,-177.473,8.107,148.837
C08915=1140.890,259.096,-69.288,-177.475,8.104,148.837
C08916=1140.895,258.848,-69.259,-177.478,8.100,148.837
C08917=1140.899,258.599,-69.232,-177.481,8.097,148.837
C08918=1140.904,258.351,-69.204,-177.484,8.094,148.837
C08919=1140.908,258.102,-69.175,-177.487,8.091,148.837
C08920=1140.913,257.854,-69.148,-177.490,8.088,148.837
C08921=1140.916,257.605,-69.120,-177.492,8.085,148.837
C08922=1140.921,257.357,-69.091,-177.495,8.082,148.837
C08923=1140.925,257.109,-69.063,-177.498,8.079,148.837
C08924=1140.929,256.861,-69.035,-177.500,8.076,148.838
C08925=1140.934,256.612,-69.007,-177.503,8.073,148.838
C08926=1140.938,256.364,-68.979,-177.506,8.070,148.838
C08927=1140.942,256.115,-68.951,-177.509,8.067,148.838
C08928=1140.947,255.867,-68.923,-177.511,8.064,148.838
C08929=1140.951,255.618,-68.895,-177.514,8.061,148.838
C08930=1140.956,255.370,-68.867,-177.517,8.058,148.838
C08931=1140.960,255.122,-68.839,-177.520,8.055,148.838
C08932=1140.965,254.873,-68.811,-177.523,8.052,148.838
C08933=1140.969,254.625,-68.783,-177.526,8.049,148.838
C08934=1140.973,254.376,-68.755,-177.528,8.046,148.838
C08935=1140.977,254.128,-68.728,-177.531,8.043,148.838
C08936=1140.982,253.879,-68.700,-177.534,8.040,148.838
C08937=1140.986,253.631,-68.672,-177.536,8.037,148.838
C08938=1140.991,253.383,-68.644,-177.539,8.034,148.838
C08939=1140.995,253.134,-68.617,-177.542,8.031,148.838
C08940=1140.999,252.886,-68.589,-177.545,8.028,148.838
C08941=1141.004,252.638,-68.560,-177.547,8.025,148.838
C08942=1141.008,252.389,-68.533,-177.550,8.022,148.838
C08943=1141.013,252.141,-68.505,-177.553,8.019,148.838
C08944=1141.017,251.892,-68.478,-177.556,8.016,148.838
C08945=1141.021,251.644,-68.450,-177.559,8.013,148.839
C08946=1141.025,251.396,-68.422,-177.561,8.010,148.838
C08947=1141.029,251.147,-68.395,-177.564,8.007,148.838
C08948=1141.034,250.899,-68.367,-177.567,8.004,148.839
C08949=1141.038,250.650,-68.340,-177.569,8.001,148.839
C08950=1141.043,250.401,-68.311,-177.572,7.998,148.839
C08951=1141.048,250.153,-68.284,-177.575,7.996,148.839
C08952=1141.052,249.905,-68.256,-177.578,7.993,148.839
C08953=1141.056,249.656,-68.229,-177.581,7.990,148.839
C08954=1141.060,249.408,-68.201,-177.583,7.987,148.839
C08955=1141.065,249.159,-68.174,-177.586,7.984,148.839
C08956=1141.069,248.910,-68.147,-177.589,7.981,148.839
C08957=1141.073,248.662,-68.119,-177.592,7.978,148.839
C08958=1141.078,248.414,-68.092,-177.595,7.974,148.839
C08959=1141.082,248.166,-68.064,-177.598,7.971,148.839
C08960=1141.086,247.917,-68.037,-177.600,7.968,148.839
C08961=1141.091,247.668,-68.010,-177.603,7.965,148.839
C08962=1141.095,247.420,-67.982,-177.606,7.962,148.839
C08963=1141.100,247.172,-67.955,-177.609,7.959,148.839
C08964=1141.104,246.923,-67.927,-177.611,7.956,148.839
C08965=1141.108,246.675,-67.900,-177.614,7.954,148.840
C08966=1141.113,246.426,-67.872,-177.617,7.951,148.840
C08967=1141.118,246.178,-67.845,-177.620,7.948,148.840
C08968=1141.122,245.929,-67.817,-177.623,7.945,148.840
C08969=1141.126,245.681,-67.790,-177.625,7.942,148.840
C08970=1141.131,245.432,-67.763,-177.628,7.939,148.840
C08971=1141.135,245.184,-67.737,-177.631,7.936,148.840
C08972=1141.139,244.936,-67.709,-177.634,7.933,148.840
C08973=1141.143,244.687,-67.681,-177.637,7.930,148.840
C08974=1141.148,244.439,-67.654,-177.639,7.928,148.840
C08975=1141.152,244.190,-67.627,-177.642,7.925,148.840
C08976=1141.157,243.942,-67.600,-177.644,7.922,148.840
C08977=1141.162,243.693,-67.573,-177.647,7.919,148.840
C08978=1141.165,243.445,-67.546,-177.650,7.916,148.841
C08979=1141.169,243.196,-67.519,-177.653,7.914,148.841
C08980=1141.174,242.948,-67.492,-177.656,7.911,148.841
C08981=1141.179,242.699,-67.464,-177.658,7.908,148.841
C08982=1141.183,242.451,-67.437,-177.661,7.905,148.841
C08983=1141.187,242.203,-67.411,-177.664,7.902,148.841
C08984=1141.191,241.953,-67.384,-177.667,7.899,148.841
C08985=1141.196,241.705,-67.356,-177.670,7.896,148.841
C08986=1141.201,241.456,-67.329,-177.672,7.893,148.841
C08987=1141.205,241.208,-67.302,-177.675,7.890,148.841
C08988=1141.209,240.960,-67.276,-177.678,7.887,148.841
C08989=1141.214,240.711,-67.249,-177.681,7.884,148.841
C08990=1141.219,240.463,-67.222,-177.684,7.881,148.841
C08991=1141.223,240.214,-67.195,-177.686,7.879,148.842
C08992=1141.227,239.965,-67.168,-177.689,7.876,148.842
C08993=1141.231,239.717,-67.141,-177.692,7.873,148.842
C08994=1141.236,239.468,-67.114,-177.695,7.870,148.842
C08995=1141.240,239.220,-67.087,-177.698,7.867,148.842
C08996=1141.244,238.972,-67.060,-177.700,7.864,148.842
C08997=1141.249,238.723,-67.034,-177.703,7.861,148.842
C08998=1141.253,238.474,-67.007,-177.706,7.858,148.842
C08999=1141.258,238.226,-66.980,-177.709,7.855,148.842
C09000=1141.263,237.977,-66.953,-177.712,7.852,148.842
C09001=1141.267,237.729,-66.927,-177.714,7.849,148.842
C09002=1141.271,237.481,-66.900,-177.717,7.847,148.842
C09003=1141.276,237.232,-66.873,-177.719,7.844,148.843
C09004=1141.280,236.983,-66.847,-177.722,7.841,148.843
C09005=1141.285,236.735,-66.820,-177.725,7.839,148.843
C09006=1141.289,236.487,-66.793,-177.728,7.836,148.843
C09007=1141.294,236.238,-66.767,-177.731,7.833,148.843
C09008=1141.298,235.989,-66.740,-177.734,7.830,148.843
C09009=1141.302,235.717,-66.711,-177.737,7.827,148.843
C09010=1141.307,235.446,-66.682,-177.740,7.823,148.843
C09011=1141.313,235.173,-66.653,-177.743,7.821,148.843
C09012=1141.317,234.902,-66.624,-177.746,7.818,148.843
C09013=1141.322,234.654,-66.597,-177.748,7.815,148.844
C09014=1141.326,234.405,-66.571,-177.751,7.812,148.844
C09015=1141.331,234.156,-66.544,-177.754,7.809,148.844
C09016=1141.335,233.908,-66.518,-177.757,7.806,148.844
C09017=1141.339,233.659,-66.491,-177.760,7.803,148.844
C09018=1141.343,233.411,-66.465,-177.763,7.800,148.844
C09019=1141.348,233.162,-66.439,-177.766,7.798,148.844
C09020=1141.352,232.913,-66.412,-177.768,7.795,148.844
C09021=1141.357,232.664,-66.386,-177.771,7.793,148.844
C09022=1141.361,232.416,-66.359,-177.773,7.790,148.845
C09023=1141.366,232.167,-66.333,-177.776,7.787,148.845
C09024=1141.370,231.919,-66.307,-177.779,7.784,148.845
C09025=1141.375,231.670,-66.280,-177.782,7.781,148.845
C09026=1141.379,231.422,-66.254,-177.785,7.778,148.845
C09027=1141.383,231.173,-66.228,-177.788,7.775,148.845
C09028=1141.388,230.924,-66.201,-177.791,7.773,148.845
C09029=1141.393,230.676,-66.176,-177.793,7.770,148.845
C09030=1141.397,230.428,-66.148,-177.796,7.767,148.845
C09031=1141.402,230.179,-66.123,-177.798,7.765,148.846
C09032=1141.405,229.931,-66.096,-177.801,7.762,148.846
C09033=1141.410,229.682,-66.070,-177.804,7.759,148.846
C09034=1141.415,229.433,-66.044,-177.807,7.756,148.846
C09035=1141.419,229.185,-66.018,-177.810,7.753,148.846
C09036=1141.424,228.935,-65.991,-177.813,7.750,148.846
C09037=1141.428,228.687,-65.966,-177.816,7.747,148.846
C09038=1141.432,228.439,-65.940,-177.819,7.745,148.846
C09039=1141.437,228.190,-65.913,-177.821,7.742,148.847
C09040=1141.441,227.941,-65.887,-177.824,7.740,148.847
C09041=1141.445,227.693,-65.861,-177.826,7.737,148.847
C09042=1141.450,227.444,-65.835,-177.829,7.734,148.847
C09043=1141.455,227.196,-65.809,-177.832,7.731,148.847
C09044=1141.459,226.947,-65.783,-177.835,7.728,148.847
C09045=1141.463,226.699,-65.757,-177.838,7.725,148.847
C09046=1141.468,226.450,-65.731,-177.840,7.723,148.847
C09047=1141.472,226.201,-65.705,-177.843,7.720,148.847
C09048=1141.477,225.953,-65.680,-177.846,7.717,148.848
C09049=1141.482,225.704,-65.654,-177.849,7.715,148.848
C09050=1141.486,225.455,-65.628,-177.852,7.712,148.848
C09051=1141.490,225.207,-65.601,-177.855,7.709,148.848
C09052=1141.495,224.958,-65.575,-177.857,7.706,148.848
C09053=1141.499,224.710,-65.550,-177.860,7.704,148.848
C09054=1141.504,224.461,-65.524,-177.863,7.701,148.848
C09055=1141.508,224.212,-65.498,-177.865,7.698,148.848
C09056=1141.512,223.963,-65.473,-177.869,7.696,148.849
C09057=1141.518,223.715,-65.447,-177.871,7.693,148.849
C09058=1141.522,223.466,-65.421,-177.874,7.690,148.849
C09059=1141.526,223.217,-65.395,-177.876,7.688,148.849
C09060=1141.531,222.969,-65.370,-177.879,7.685,148.849
C09061=1141.535,222.720,-65.344,-177.882,7.682,148.849
C09062=1141.539,222.472,-65.318,-177.885,7.679,148.850
C09063=1141.544,222.223,-65.292,-177.888,7.676,148.850
C09064=1141.548,221.975,-65.267,-177.891,7.673,148.850
C09065=1141.553,221.726,-65.241,-177.893,7.671,148.850
C09066=1141.557,221.477,-65.216,-177.896,7.669,148.850
C09067=1141.562,221.229,-65.190,-177.899,7.666,148.850
C09068=1141.567,220.980,-65.164,-177.902,7.663,148.850
C09069=1141.571,220.731,-65.138,-177.905,7.660,148.850
C09070=1141.576,220.483,-65.113,-177.908,7.657,148.851
C09071=1141.580,220.234,-65.087,-177.910,7.655,148.851
C09072=1141.584,219.985,-65.061,-177.913,7.653,148.851
C09073=1141.589,219.737,-65.037,-177.916,7.650,148.851
C09074=1141.594,219.488,-65.011,-177.919,7.647,148.851
C09075=1141.598,219.239,-64.985,-177.921,7.644,148.851
C09076=1141.603,218.991,-64.960,-177.924,7.642,148.852
C09077=1141.607,218.742,-64.934,-177.927,7.639,148.852
C09078=1141.611,218.493,-64.908,-177.930,7.636,148.852
C09079=1141.615,218.245,-64.884,-177.933,7.633,148.852
C09080=1141.620,217.996,-64.858,-177.936,7.631,148.852
C09081=1141.624,217.747,-64.833,-177.938,7.629,148.852
C09082=1141.629,217.499,-64.807,-177.941,7.626,148.852
C09083=1141.633,217.250,-64.782,-177.944,7.623,148.853
C09084=1141.638,217.002,-64.757,-177.947,7.620,148.853
C09085=1141.642,216.753,-64.731,-177.950,7.617,148.853
C09086=1141.647,216.503,-64.706,-177.952,7.615,148.853
C09087=1141.652,216.255,-64.681,-177.955,7.612,148.853
C09088=1141.656,216.007,-64.655,-177.958,7.610,148.853
C09089=1141.660,215.758,-64.631,-177.961,7.607,148.854
C09090=1141.665,215.509,-64.605,-177.963,7.605,148.854
C09091=1141.669,215.261,-64.580,-177.966,7.602,148.854
C09092=1141.674,215.012,-64.555,-177.969,7.599,148.854
C09093=1141.678,214.763,-64.529,-177.972,7.596,148.854
C09094=1141.683,214.515,-64.503,-177.975,7.594,148.854
C09095=1141.687,214.266,-64.479,-177.977,7.591,148.854
C09096=1141.692,214.018,-64.454,-177.980,7.589,148.855
C09097=1141.696,213.768,-64.429,-177.983,7.586,148.855
C09098=1141.701,213.520,-64.403,-177.986,7.583,148.855
C09099=1141.705,213.271,-64.378,-177.988,7.581,148.855
C09100=1141.710,213.023,-64.353,-177.991,7.578,148.855
C09101=1141.714,212.774,-64.328,-177.994,7.575,148.855
C09102=1141.719,212.525,-64.303,-177.997,7.573,148.856
C09103=1141.723,212.276,-64.278,-178.000,7.571,148.856
C09104=1141.727,212.028,-64.253,-178.002,7.568,148.856
C09105=1141.732,211.779,-64.228,-178.005,7.565,148.856
C09106=1141.737,211.530,-64.203,-178.008,7.562,148.856
C09107=1141.741,211.281,-64.178,-178.011,7.560,148.857
C09108=1141.746,211.033,-64.154,-178.013,7.557,148.857
C09109=1141.750,210.784,-64.128,-178.017,7.555,148.857
C09110=1141.755,210.535,-64.103,-178.020,7.552,148.857
C09111=1141.760,210.287,-64.079,-178.022,7.550,148.857
C09112=1141.764,210.038,-64.053,-178.025,7.547,148.857
C09113=1141.768,209.767,-64.026,-178.028,7.544,148.858
C09114=1141.773,209.497,-64.000,-178.031,7.542,148.858
C09115=1141.779,209.226,-63.972,-178.034,7.539,148.858
C09116=1141.784,208.956,-63.945,-178.037,7.536,148.858
C09117=1141.788,208.707,-63.921,-178.040,7.533,148.858
C09118=1141.793,208.458,-63.896,-178.043,7.531,148.859
C09119=1141.798,208.210,-63.871,-178.045,7.528,148.859
C09120=1141.801,207.961,-63.846,-178.048,7.526,148.859
C09121=1141.807,207.712,-63.822,-178.051,7.523,148.859
C09122=1141.810,207.463,-63.797,-178.054,7.520,148.859
C09123=1141.815,207.215,-63.772,-178.057,7.518,148.860
C09124=1141.820,206.966,-63.747,-178.059,7.515,148.860
C09125=1141.824,206.717,-63.723,-178.062,7.513,148.860
C09126=1141.829,206.468,-63.698,-178.065,7.511,148.860
C09127=1141.834,206.220,-63.674,-178.068,7.508,148.860
C09128=1141.838,205.970,-63.649,-178.070,7.505,148.860
C09129=1141.843,205.722,-63.625,-178.074,7.502,148.861
C09130=1141.847,205.473,-63.599,-178.076,7.500,148.861
C09131=1141.851,205.225,-63.575,-178.079,7.497,148.861
C09132=1141.856,204.976,-63.550,-178.082,7.495,148.861
C09133=1141.860,204.727,-63.526,-178.084,7.493,148.861
C09134=1141.865,204.478,-63.501,-178.088,7.490,148.862
C09135=1141.870,204.230,-63.477,-178.090,7.487,148.862
C09136=1141.875,203.981,-63.452,-178.093,7.485,148.862
C09137=1141.879,203.732,-63.428,-178.096,7.483,148.862
C09138=1141.884,203.483,-63.403,-178.099,7.480,148.862
C09139=1141.888,203.235,-63.379,-178.101,7.478,148.862
C09140=1141.892,202.986,-63.355,-178.104,7.475,148.863
C09141=1141.897,202.737,-63.330,-178.107,7.472,148.863
C09142=1141.901,202.488,-63.306,-178.110,7.471,148.863
C09143=1141.906,202.239,-63.281,-178.112,7.468,148.863
C09144=1141.910,201.991,-63.257,-178.115,7.465,148.863
C09145=1141.915,201.742,-63.233,-178.118,7.463,148.864
